LIN {X 0,Y 408.428,Z 752.813,A -85,B 0,C 180,E1 10680.84,E2 10680.84} C_VEL
LIN {X 0,Y 404.021,Z 784.174,A -85,B 0,C 180,E1 10684.706,E2 10684.706} C_VEL
LIN {X 0,Y 400.788,Z 809.614,A -85,B 0,C 180,E1 10688.967,E2 10688.967} C_VEL
LIN {X 0,Y 398.664,Z 830.61,A -85,B 0,C 180,E1 10693.733,E2 10693.733} C_VEL
LIN {X 0,Y 397.715,Z 845.382,A -85,B 0,C 180,E1 10698.469,E2 10698.469} C_VEL
LIN {X 0,Y 397.631,Z 847.747,A -85,B 0,C 180,E1 10699.458,E2 10699.458} C_VEL
LIN {X 0,Y 395.083,Z 851.309,A -85,B 0,C 180,E1 10701.251,E2 10701.251} C_VEL
LIN {X 0,Y 389.791,Z 854.941,A -85,B 0,C 180,E1 10704.007,E2 10704.007} C_VEL
LIN {X 0,Y 389.709,Z 855.317,A -85,B 0,C 180,E1 10704.327,E2 10704.327} C_VEL
LIN {X 0,Y 389.668,Z 858.175,A -85,B 0,C 180,E1 10707.771,E2 10707.771} C_VEL
LIN {X 0,Y 389.693,Z 858.182,A -85,B 0,C 180,E1 10712.225,E2 10712.225} C_VEL
LIN {X 0,Y 389.728,Z 854.056,A -85,B 0,C 180,E1 10716.691,E2 10716.691} C_VEL
LIN {X 0,Y 389.922,Z 844.142,A -85,B 0,C 180,E1 10721.76,E2 10721.76} C_VEL
LIN {X 0,Y 390.93,Z 828.247,A -85,B 0,C 180,E1 10726.884,E2 10726.884} C_VEL
LIN {X 0,Y 393.21,Z 806.828,A -85,B 0,C 180,E1 10731.751,E2 10731.751} C_VEL
LIN {X 0,Y 397.092,Z 778.974,A -85,B 0,C 180,E1 10736.349,E2 10736.349} C_VEL
LIN {X 0,Y 401.785,Z 748.417,A -85,B 0,C 180,E1 10740.034,E2 10740.034} C_VEL
LIN {X 0,Y 406.818,Z 713.375,A -85,B 0,C 180,E1 10743.071,E2 10743.071} C_VEL
LIN {X 0,Y 411.253,Z 676.937,A -85,B 0,C 180,E1 10745.194,E2 10745.194} C_VEL
LIN {X 0,Y 413.797,Z 641.889,A -85,B 0,C 180,E1 10746.487,E2 10746.487} C_VEL
LIN {X 0,Y 400.605,Z 608.761,A -85,B 0,C 180,E1 10748.579,E2 10748.579} C_VEL
LIN {X 0,Y 387.28,Z 580.66,A -85,B 0,C 180,E1 10750.746,E2 10750.746} C_VEL
LIN {X 0,Y 387.242,Z 580.66,A -85,B 0,C 180,E1 10757.972,E2 10757.972} C_VEL
LIN {X 0,Y 387.329,Z 580.66,A -85,B 0,C 180,E1 10765.168,E2 10765.168} C_VEL
LIN {X 0,Y 387.521,Z 580.66,A -85,B 0,C 180,E1 10772.048,E2 10772.048} C_VEL
LIN {X 0,Y 387.806,Z 580.66,A -85,B 0,C 180,E1 10779.543,E2 10779.543} C_VEL
LIN {X 0,Y 387.952,Z 580.66,A -85,B 0,C 180,E1 10786.464,E2 10786.464} C_VEL
LIN {X 0,Y 388.392,Z 580.66,A -85,B 0,C 180,E1 10793.29,E2 10793.29} C_VEL
LIN {X 0,Y 388.731,Z 580.66,A -85,B 0,C 180,E1 10800.006,E2 10800.006} C_VEL
LIN {X 0,Y 388.325,Z 580.66,A -85,B 0,C 180,E1 10806.723,E2 10806.723} C_VEL
LIN {X 0,Y 388.031,Z 580.66,A -85,B 0,C 180,E1 10813.546,E2 10813.546} C_VEL
LIN {X 0,Y 387.797,Z 580.66,A -85,B 0,C 180,E1 10820.578,E2 10820.578} C_VEL
LIN {X 0,Y 387.538,Z 580.66,A -85,B 0,C 180,E1 10827.964,E2 10827.964} C_VEL
LIN {X 0,Y 387.36,Z 580.66,A -85,B 0,C 180,E1 10835.902,E2 10835.902} C_VEL
LIN {X 0,Y 387.152,Z 580.66,A -85,B 0,C 180,E1 10842.013,E2 10842.013} C_VEL
LIN {X 0,Y 387.17,Z 580.66,A -85,B 0,C 180,E1 10848.337,E2 10848.337} C_VEL
LIN {X 0,Y 387.501,Z 581.204,A -85,B 0,C 180,E1 10855.685,E2 10855.685} C_VEL
LIN {X 0,Y 400.111,Z 612.182,A -85,B 0,C 180,E1 10858.859,E2 10858.859} C_VEL
LIN {X 0,Y 408.135,Z 640.7,A -85,B 0,C 180,E1 10862.182,E2 10862.182} C_VEL
LIN {X 0,Y 408.327,Z 648.198,A -85,B 0,C 180,E1 10863.018,E2 10863.018} C_VEL
LIN {X 0,Y 403.521,Z 675.315,A -85,B 0,C 180,E1 10866.233,E2 10866.233} C_VEL
LIN {X 0,Y 399.051,Z 697.721,A -85,B 0,C 180,E1 10870.036,E2 10870.036} C_VEL
LIN {X 0,Y 395.127,Z 716.014,A -85,B 0,C 180,E1 10874.444,E2 10874.444} C_VEL
LIN {X 0,Y 392.367,Z 729.811,A -85,B 0,C 180,E1 10879.554,E2 10879.554} C_VEL
LIN {X 0,Y 391.047,Z 737.35,A -85,B 0,C 180,E1 10884.448,E2 10884.448} C_VEL
LIN {X 0,Y 390.565,Z 740.223,A -85,B 0,C 180,E1 10890.002,E2 10890.002} C_VEL
LIN {X 0,Y 391.048,Z 737.251,A -85,B 0,C 180,E1 10895.557,E2 10895.557} C_VEL
LIN {X 0,Y 392.34,Z 729.704,A -85,B 0,C 180,E1 10900.402,E2 10900.402} C_VEL
LIN {X 0,Y 394.76,Z 717.487,A -85,B 0,C 180,E1 10905.006,E2 10905.006} C_VEL
LIN {X 0,Y 398.476,Z 699.978,A -85,B 0,C 180,E1 10909.42,E2 10909.42} C_VEL
LIN {X 0,Y 402.996,Z 677.934,A -85,B 0,C 180,E1 10913.277,E2 10913.277} C_VEL
LIN {X 0,Y 407.688,Z 652.329,A -85,B 0,C 180,E1 10916.467,E2 10916.467} C_VEL
LIN {X 0,Y 408.513,Z 642.184,A -85,B 0,C 180,E1 10917.525,E2 10917.525} C_VEL
LIN {X 0,Y 400.672,Z 614.076,A -85,B 0,C 180,E1 10920.832,E2 10920.832} C_VEL
LIN {X 0,Y 388.716,Z 584.955,A -85,B 0,C 180,E1 10923.905,E2 10923.905} C_VEL
LIN {X 0,Y 387.379,Z 580.66,A -85,B 0,C 180,E1 10924.312,E2 10924.312} C_VEL
LIN {X 0,Y 387.223,Z 580.66,A -85,B 0,C 180,E1 10931.661,E2 10931.661} C_VEL
LIN {X 0,Y 387.212,Z 580.66,A -85,B 0,C 180,E1 10938.331,E2 10938.331} C_VEL
LIN {X 0,Y 387.234,Z 580.66,A -85,B 0,C 180,E1 10945.195,E2 10945.195} C_VEL
LIN {X 0,Y 387.521,Z 580.66,A -85,B 0,C 180,E1 10952.034,E2 10952.034} C_VEL
LIN {X 0,Y 387.844,Z 580.66,A -85,B 0,C 180,E1 10959.54,E2 10959.54} C_VEL
LIN {X 0,Y 387.884,Z 580.66,A -85,B 0,C 180,E1 10966.449,E2 10966.449} C_VEL
LIN {X 0,Y 388.423,Z 580.66,A -85,B 0,C 180,E1 10973.278,E2 10973.278} C_VEL
LIN {X 0,Y 388.731,Z 580.66,A -85,B 0,C 180,E1 10979.994,E2 10979.994} C_VEL
LIN {X 0,Y 388.342,Z 580.66,A -85,B 0,C 180,E1 10986.71,E2 10986.71} C_VEL
LIN {X 0,Y 388.039,Z 580.66,A -85,B 0,C 180,E1 10993.532,E2 10993.532} C_VEL
LIN {X 0,Y 387.8,Z 580.66,A -85,B 0,C 180,E1 11000.565,E2 11000.565} C_VEL
LIN {X 0,Y 387.52,Z 580.66,A -85,B 0,C 180,E1 11007.952,E2 11007.952} C_VEL
LIN {X 0,Y 387.321,Z 580.66,A -85,B 0,C 180,E1 11014.824,E2 11014.824} C_VEL
LIN {X 0,Y 387.199,Z 580.66,A -85,B 0,C 180,E1 11022.015,E2 11022.015} C_VEL
LIN {X 0,Y 387.338,Z 580.66,A -85,B 0,C 180,E1 11029.326,E2 11029.326} C_VEL
LIN {X 0,Y 395.978,Z 599.127,A -85,B 0,C 180,E1 11030.728,E2 11030.728} C_VEL
LIN {X 0,Y 411.678,Z 635.468,A -85,B 0,C 180,E1 11033.137,E2 11033.137} C_VEL
LIN {X 0,Y 414.185,Z 645.901,A -85,B 0,C 180,E1 11033.687,E2 11033.687} C_VEL
LIN {X 0,Y 410.314,Z 684.949,A -85,B 0,C 180,E1 11035.193,E2 11035.193} C_VEL
LIN {X 0,Y 405.769,Z 720.46,A -85,B 0,C 180,E1 11037.462,E2 11037.462} C_VEL
LIN {X 0,Y 400.817,Z 754.356,A -85,B 0,C 180,E1 11040.588,E2 11040.588} C_VEL
LIN {X 0,Y 396.311,Z 784.649,A -85,B 0,C 180,E1 11044.482,E2 11044.482} C_VEL
LIN {X 0,Y 392.955,Z 809.701,A -85,B 0,C 180,E1 11048.823,E2 11048.823} C_VEL
LIN {X 0,Y 390.795,Z 830.377,A -85,B 0,C 180,E1 11053.685,E2 11053.685} C_VEL
LIN {X 0,Y 389.827,Z 845.492,A -85,B 0,C 180,E1 11058.8,E2 11058.8} C_VEL
LIN {X 0,Y 389.735,Z 854.049,A -85,B 0,C 180,E1 11063.305,E2 11063.305} C_VEL
LIN {X 0,Y 389.709,Z 855.317,A -85,B 0,C 180,E1 11064.327,E2 11064.327} C_VEL
LIN {X 0,Y 387.19,Z 856.88,A -85,B 0,C 180,E1 11066.212,E2 11066.212} C_VEL
LIN {X 0,Y 381.917,Z 857.427,A -85,B 0,C 180,E1 11069.077,E2 11069.077} C_VEL
LIN {X 0,Y 381.856,Z 857.421,A -85,B 0,C 180,E1 11069.408,E2 11069.408} C_VEL
LIN {X 0,Y 381.884,Z 855.425,A -85,B 0,C 180,E1 11074.546,E2 11074.546} C_VEL
LIN {X 0,Y 381.91,Z 849.075,A -85,B 0,C 180,E1 11079.122,E2 11079.122} C_VEL
LIN {X 0,Y 382.441,Z 836.232,A -85,B 0,C 180,E1 11084.44,E2 11084.44} C_VEL
LIN {X 0,Y 384.2,Z 817.301,A -85,B 0,C 180,E1 11089.683,E2 11089.683} C_VEL
LIN {X 0,Y 387.498,Z 792.723,A -85,B 0,C 180,E1 11094.526,E2 11094.526} C_VEL
LIN {X 0,Y 391.958,Z 763.881,A -85,B 0,C 180,E1 11098.711,E2 11098.711} C_VEL
LIN {X 0,Y 397.257,Z 730.096,A -85,B 0,C 180,E1 11102.244,E2 11102.244} C_VEL
LIN {X 0,Y 402.324,Z 695.108,A -85,B 0,C 180,E1 11104.795,E2 11104.795} C_VEL
LIN {X 0,Y 406.63,Z 657.105,A -85,B 0,C 180,E1 11106.562,E2 11106.562} C_VEL
LIN {X 0,Y 407.134,Z 644.103,A -85,B 0,C 180,E1 11107.017,E2 11107.017} C_VEL
LIN {X 0,Y 394.189,Z 611.589,A -85,B 0,C 180,E1 11109.175,E2 11109.175} C_VEL
LIN {X 0,Y 379.324,Z 580.66,A -85,B 0,C 180,E1 11111.638,E2 11111.638} C_VEL
LIN {X 0,Y 379.285,Z 580.66,A -85,B 0,C 180,E1 11117.274,E2 11117.274} C_VEL
LIN {X 0,Y 379.32,Z 580.66,A -85,B 0,C 180,E1 11123.23,E2 11123.23} C_VEL
LIN {X 0,Y 379.421,Z 580.66,A -85,B 0,C 180,E1 11128.759,E2 11128.759} C_VEL
LIN {X 0,Y 379.685,Z 580.66,A -85,B 0,C 180,E1 11136.506,E2 11136.506} C_VEL
LIN {X 0,Y 379.941,Z 580.66,A -85,B 0,C 180,E1 11143.809,E2 11143.809} C_VEL
LIN {X 0,Y 380.271,Z 580.66,A -85,B 0,C 180,E1 11150.843,E2 11150.843} C_VEL
LIN {X 0,Y 380.781,Z 580.66,A -85,B 0,C 180,E1 11157.728,E2 11157.728} C_VEL
LIN {X 0,Y 380.595,Z 580.66,A -85,B 0,C 180,E1 11164.57,E2 11164.57} C_VEL
LIN {X 0,Y 380.168,Z 580.66,A -85,B 0,C 180,E1 11171.492,E2 11171.492} C_VEL
LIN {X 0,Y 379.949,Z 580.66,A -85,B 0,C 180,E1 11178.596,E2 11178.596} C_VEL
LIN {X 0,Y 379.641,Z 580.66,A -85,B 0,C 180,E1 11186.027,E2 11186.027} C_VEL
LIN {X 0,Y 379.449,Z 580.66,A -85,B 0,C 180,E1 11193.967,E2 11193.967} C_VEL
LIN {X 0,Y 379.2,Z 580.66,A -85,B 0,C 180,E1 11200.662,E2 11200.662} C_VEL
LIN {X 0,Y 379.165,Z 580.66,A -85,B 0,C 180,E1 11207.252,E2 11207.252} C_VEL
LIN {X 0,Y 379.517,Z 580.66,A -85,B 0,C 180,E1 11214.699,E2 11214.699} C_VEL
LIN {X 0,Y 392.526,Z 612.432,A -85,B 0,C 180,E1 11218.068,E2 11218.068} C_VEL
LIN {X 0,Y 400.461,Z 640.281,A -85,B 0,C 180,E1 11221.385,E2 11221.385} C_VEL
LIN {X 0,Y 401.55,Z 648.886,A -85,B 0,C 180,E1 11222.445,E2 11222.445} C_VEL
LIN {X 0,Y 396.58,Z 675.766,A -85,B 0,C 180,E1 11225.66,E2 11225.66} C_VEL
LIN {X 0,Y 391.704,Z 698.972,A -85,B 0,C 180,E1 11229.645,E2 11229.645} C_VEL
LIN {X 0,Y 387.601,Z 717.228,A -85,B 0,C 180,E1 11234.134,E2 11234.134} C_VEL
LIN {X 0,Y 384.971,Z 729.548,A -85,B 0,C 180,E1 11238.662,E2 11238.662} C_VEL
LIN {X 0,Y 383.57,Z 737.237,A -85,B 0,C 180,E1 11243.201,E2 11243.201} C_VEL
LIN {X 0,Y 382.888,Z 740.919,A -85,B 0,C 180,E1 11247.736,E2 11247.736} C_VEL
LIN {X 0,Y 383,Z 740.86,A -85,B 0,C 180,E1 11252.268,E2 11252.268} C_VEL
LIN {X 0,Y 383.558,Z 737.112,A -85,B 0,C 180,E1 11256.803,E2 11256.803} C_VEL
LIN {X 0,Y 385.296,Z 728.075,A -85,B 0,C 180,E1 11261.908,E2 11261.908} C_VEL
LIN {X 0,Y 388.46,Z 713.123,A -85,B 0,C 180,E1 11266.937,E2 11266.937} C_VEL
LIN {X 0,Y 392.989,Z 692.75,A -85,B 0,C 180,E1 11271.471,E2 11271.471} C_VEL
LIN {X 0,Y 397.941,Z 668.776,A -85,B 0,C 180,E1 11275.194,E2 11275.194} C_VEL
LIN {X 0,Y 401.712,Z 645.578,A -85,B 0,C 180,E1 11277.822,E2 11277.822} C_VEL
LIN {X 0,Y 394.415,Z 618.304,A -85,B 0,C 180,E1 11281.162,E2 11281.162} C_VEL
LIN {X 0,Y 383.249,Z 590.025,A -85,B 0,C 180,E1 11284.285,E2 11284.285} C_VEL
LIN {X 0,Y 379.427,Z 580.66,A -85,B 0,C 180,E1 11285.311,E2 11285.311} C_VEL
LIN {X 0,Y 379.232,Z 580.66,A -85,B 0,C 180,E1 11292.745,E2 11292.745} C_VEL
LIN {X 0,Y 379.221,Z 580.66,A -85,B 0,C 180,E1 11300.29,E2 11300.29} C_VEL
LIN {X 0,Y 379.372,Z 580.66,A -85,B 0,C 180,E1 11306.942,E2 11306.942} C_VEL
LIN {X 0,Y 379.642,Z 580.66,A -85,B 0,C 180,E1 11313.973,E2 11313.973} C_VEL
LIN {X 0,Y 379.927,Z 580.66,A -85,B 0,C 180,E1 11321.403,E2 11321.403} C_VEL
LIN {X 0,Y 380.06,Z 580.66,A -85,B 0,C 180,E1 11328.504,E2 11328.504} C_VEL
LIN {X 0,Y 380.542,Z 580.66,A -85,B 0,C 180,E1 11335.43,E2 11335.43} C_VEL
LIN {X 0,Y 380.829,Z 580.66,A -85,B 0,C 180,E1 11339.994,E2 11339.994} C_VEL
LIN {X 0,Y 380.431,Z 580.66,A -85,B 0,C 180,E1 11346.851,E2 11346.851} C_VEL
LIN {X 0,Y 380.096,Z 580.66,A -85,B 0,C 180,E1 11353.821,E2 11353.821} C_VEL
LIN {X 0,Y 379.823,Z 580.66,A -85,B 0,C 180,E1 11361.017,E2 11361.017} C_VEL
LIN {X 0,Y 379.537,Z 580.66,A -85,B 0,C 180,E1 11368.641,E2 11368.641} C_VEL
LIN {X 0,Y 379.402,Z 580.66,A -85,B 0,C 180,E1 11373.957,E2 11373.957} C_VEL
LIN {X 0,Y 379.234,Z 580.66,A -85,B 0,C 180,E1 11380.661,E2 11380.661} C_VEL
LIN {X 0,Y 379.354,Z 580.66,A -85,B 0,C 180,E1 11388.357,E2 11388.357} C_VEL
LIN {X 0,Y 402.366,Z 630.289,A -85,B 0,C 180,E1 11392.12,E2 11392.12} C_VEL
LIN {X 0,Y 407.505,Z 646.855,A -85,B 0,C 180,E1 11393.118,E2 11393.118} C_VEL
LIN {X 0,Y 403.389,Z 685.45,A -85,B 0,C 180,E1 11394.662,E2 11394.662} C_VEL
LIN {X 0,Y 398.627,Z 720.792,A -85,B 0,C 180,E1 11396.983,E2 11396.983} C_VEL
LIN {X 0,Y 393.277,Z 755.365,A -85,B 0,C 180,E1 11400.285,E2 11400.285} C_VEL
LIN {X 0,Y 388.564,Z 785.437,A -85,B 0,C 180,E1 11404.295,E2 11404.295} C_VEL
LIN {X 0,Y 384.994,Z 811.22,A -85,B 0,C 180,E1 11408.97,E2 11408.97} C_VEL
LIN {X 0,Y 382.809,Z 831.032,A -85,B 0,C 180,E1 11413.925,E2 11413.925} C_VEL
LIN {X 0,Y 381.942,Z 845.542,A -85,B 0,C 180,E1 11419.145,E2 11419.145} C_VEL
LIN {X 0,Y 381.903,Z 854.237,A -85,B 0,C 180,E1 11424.31,E2 11424.31} C_VEL
LIN {X 0,Y 381.856,Z 857.421,A -85,B 0,C 180,E1 11429.408,E2 11429.408} C_VEL
LIN {X 0,Y 379.393,Z 857.009,A -85,B 0,C 180,E1 11431.343,E2 11431.343} C_VEL
LIN {X 0,Y 374.108,Z 854.57,A -85,B 0,C 180,E1 11434.246,E2 11434.246} C_VEL
LIN {X 0,Y 374.055,Z 854.268,A -85,B 0,C 180,E1 11434.584,E2 11434.584} C_VEL
LIN {X 0,Y 374.058,Z 847.85,A -85,B 0,C 180,E1 11439.315,E2 11439.315} C_VEL
LIN {X 0,Y 374.602,Z 835.485,A -85,B 0,C 180,E1 11444.569,E2 11444.569} C_VEL
LIN {X 0,Y 376.472,Z 816.475,A -85,B 0,C 180,E1 11449.987,E2 11449.987} C_VEL
LIN {X 0,Y 380.035,Z 791.361,A -85,B 0,C 180,E1 11455.04,E2 11455.04} C_VEL
LIN {X 0,Y 384.927,Z 761.75,A -85,B 0,C 180,E1 11459.388,E2 11459.388} C_VEL
LIN {X 0,Y 390.339,Z 728.546,A -85,B 0,C 180,E1 11462.887,E2 11462.887} C_VEL
LIN {X 0,Y 395.823,Z 692.6,A -85,B 0,C 180,E1 11465.513,E2 11465.513} C_VEL
LIN {X 0,Y 400.25,Z 654.842,A -85,B 0,C 180,E1 11467.243,E2 11467.243} C_VEL
LIN {X 0,Y 400.059,Z 644.9,A -85,B 0,C 180,E1 11467.658,E2 11467.658} C_VEL
LIN {X 0,Y 386.799,Z 612.231,A -85,B 0,C 180,E1 11469.957,E2 11469.957} C_VEL
LIN {X 0,Y 371.426,Z 581.632,A -85,B 0,C 180,E1 11472.55,E2 11472.55} C_VEL
LIN {X 0,Y 371.358,Z 580.66,A -85,B 0,C 180,E1 11472.799,E2 11472.799} C_VEL
LIN {X 0,Y 371.392,Z 580.66,A -85,B 0,C 180,E1 11479.296,E2 11479.296} C_VEL
LIN {X 0,Y 371.383,Z 580.66,A -85,B 0,C 180,E1 11485.206,E2 11485.206} C_VEL
LIN {X 0,Y 371.544,Z 580.66,A -85,B 0,C 180,E1 11490.733,E2 11490.733} C_VEL
LIN {X 0,Y 371.713,Z 580.66,A -85,B 0,C 180,E1 11495.971,E2 11495.971} C_VEL
LIN {X 0,Y 371.943,Z 580.66,A -85,B 0,C 180,E1 11501.002,E2 11501.002} C_VEL
LIN {X 0,Y 372.142,Z 580.66,A -85,B 0,C 180,E1 11508.27,E2 11508.27} C_VEL
LIN {X 0,Y 372.599,Z 580.66,A -85,B 0,C 180,E1 11515.345,E2 11515.345} C_VEL
LIN {X 0,Y 372.928,Z 580.66,A -85,B 0,C 180,E1 11520.006,E2 11520.006} C_VEL
LIN {X 0,Y 372.487,Z 580.66,A -85,B 0,C 180,E1 11527.011,E2 11527.011} C_VEL
LIN {X 0,Y 372.146,Z 580.66,A -85,B 0,C 180,E1 11534.135,E2 11534.135} C_VEL
LIN {X 0,Y 371.841,Z 580.66,A -85,B 0,C 180,E1 11541.504,E2 11541.504} C_VEL
LIN {X 0,Y 371.647,Z 580.66,A -85,B 0,C 180,E1 11546.63,E2 11546.63} C_VEL
LIN {X 0,Y 371.531,Z 580.66,A -85,B 0,C 180,E1 11551.997,E2 11551.997} C_VEL
LIN {X 0,Y 371.314,Z 580.66,A -85,B 0,C 180,E1 11559.224,E2 11559.224} C_VEL
LIN {X 0,Y 371.241,Z 580.66,A -85,B 0,C 180,E1 11566.111,E2 11566.111} C_VEL
LIN {X 0,Y 371.502,Z 580.66,A -85,B 0,C 180,E1 11573.68,E2 11573.68} C_VEL
LIN {X 0,Y 385.033,Z 612.913,A -85,B 0,C 180,E1 11577.267,E2 11577.267} C_VEL
LIN {X 0,Y 393.296,Z 641.778,A -85,B 0,C 180,E1 11580.814,E2 11580.814} C_VEL
LIN {X 0,Y 394.422,Z 651.706,A -85,B 0,C 180,E1 11582.07,E2 11582.07} C_VEL
LIN {X 0,Y 389.345,Z 677.782,A -85,B 0,C 180,E1 11585.292,E2 11585.292} C_VEL
LIN {X 0,Y 384.395,Z 700.217,A -85,B 0,C 180,E1 11589.24,E2 11589.24} C_VEL
LIN {X 0,Y 380.07,Z 718.443,A -85,B 0,C 180,E1 11593.811,E2 11593.811} C_VEL
LIN {X 0,Y 376.989,Z 732.207,A -85,B 0,C 180,E1 11599.12,E2 11599.12} C_VEL
LIN {X 0,Y 375.503,Z 739.727,A -85,B 0,C 180,E1 11604.217,E2 11604.217} C_VEL
LIN {X 0,Y 374.961,Z 742.594,A -85,B 0,C 180,E1 11610.002,E2 11610.002} C_VEL
LIN {X 0,Y 375.362,Z 740.704,A -85,B 0,C 180,E1 11614.629,E2 11614.629} C_VEL
LIN {X 0,Y 376.741,Z 733.236,A -85,B 0,C 180,E1 11620.241,E2 11620.241} C_VEL
LIN {X 0,Y 379.285,Z 721.716,A -85,B 0,C 180,E1 11625.04,E2 11625.04} C_VEL
LIN {X 0,Y 383.507,Z 703.74,A -85,B 0,C 180,E1 11629.91,E2 11629.91} C_VEL
LIN {X 0,Y 388.481,Z 681.784,A -85,B 0,C 180,E1 11633.988,E2 11633.988} C_VEL
LIN {X 0,Y 393.842,Z 655.099,A -85,B 0,C 180,E1 11637.474,E2 11637.474} C_VEL
LIN {X 0,Y 394.48,Z 647.059,A -85,B 0,C 180,E1 11638.38,E2 11638.38} C_VEL
LIN {X 0,Y 387.275,Z 619.827,A -85,B 0,C 180,E1 11641.82,E2 11641.82} C_VEL
LIN {X 0,Y 376.077,Z 591.221,A -85,B 0,C 180,E1 11645.09,E2 11645.09} C_VEL
LIN {X 0,Y 371.464,Z 580.66,A -85,B 0,C 180,E1 11646.202,E2 11646.202} C_VEL
LIN {X 0,Y 371.317,Z 580.66,A -85,B 0,C 180,E1 11653.884,E2 11653.884} C_VEL
LIN {X 0,Y 371.291,Z 580.66,A -85,B 0,C 180,E1 11660.787,E2 11660.787} C_VEL
LIN {X 0,Y 371.46,Z 580.66,A -85,B 0,C 180,E1 11667.996,E2 11667.996} C_VEL
LIN {X 0,Y 371.689,Z 580.66,A -85,B 0,C 180,E1 11673.66,E2 11673.66} C_VEL
LIN {X 0,Y 371.964,Z 580.66,A -85,B 0,C 180,E1 11680.989,E2 11680.989} C_VEL
LIN {X 0,Y 372.117,Z 580.66,A -85,B 0,C 180,E1 11688.255,E2 11688.255} C_VEL
LIN {X 0,Y 372.63,Z 580.66,A -85,B 0,C 180,E1 11695.332,E2 11695.332} C_VEL
LIN {X 0,Y 372.927,Z 580.66,A -85,B 0,C 180,E1 11699.994,E2 11699.994} C_VEL
LIN {X 0,Y 372.504,Z 580.66,A -85,B 0,C 180,E1 11706.997,E2 11706.997} C_VEL
LIN {X 0,Y 372.153,Z 580.66,A -85,B 0,C 180,E1 11714.122,E2 11714.122} C_VEL
LIN {X 0,Y 371.848,Z 580.66,A -85,B 0,C 180,E1 11721.49,E2 11721.49} C_VEL
LIN {X 0,Y 371.664,Z 580.66,A -85,B 0,C 180,E1 11726.615,E2 11726.615} C_VEL
LIN {X 0,Y 371.492,Z 580.66,A -85,B 0,C 180,E1 11731.986,E2 11731.986} C_VEL
LIN {X 0,Y 371.293,Z 580.66,A -85,B 0,C 180,E1 11739.213,E2 11739.213} C_VEL
LIN {X 0,Y 371.346,Z 580.66,A -85,B 0,C 180,E1 11746.12,E2 11746.12} C_VEL
LIN {X 0,Y 371.418,Z 581.101,A -85,B 0,C 180,E1 11747.451,E2 11747.451} C_VEL
LIN {X 0,Y 394.617,Z 629.646,A -85,B 0,C 180,E1 11751.327,E2 11751.327} C_VEL
LIN {X 0,Y 400.779,Z 648.749,A -85,B 0,C 180,E1 11752.559,E2 11752.559} C_VEL
LIN {X 0,Y 396.475,Z 686.244,A -85,B 0,C 180,E1 11754.129,E2 11754.129} C_VEL
LIN {X 0,Y 391.426,Z 721.858,A -85,B 0,C 180,E1 11756.546,E2 11756.546} C_VEL
LIN {X 0,Y 385.878,Z 755.621,A -85,B 0,C 180,E1 11759.883,E2 11759.883} C_VEL
LIN {X 0,Y 381.114,Z 784.292,A -85,B 0,C 180,E1 11763.796,E2 11763.796} C_VEL
LIN {X 0,Y 377.281,Z 810.188,A -85,B 0,C 180,E1 11768.588,E2 11768.588} C_VEL
LIN {X 0,Y 375.061,Z 829.759,A -85,B 0,C 180,E1 11773.584,E2 11773.584} C_VEL
LIN {X 0,Y 374.088,Z 844.302,A -85,B 0,C 180,E1 11778.914,E2 11778.914} C_VEL
LIN {X 0,Y 374.059,Z 851.627,A -85,B 0,C 180,E1 11783.023,E2 11783.023} C_VEL
LIN {X 0,Y 374.022,Z 855.793,A -85,B 0,C 180,E1 11787.678,E2 11787.678} C_VEL
LIN {X 0,Y 374.046,Z 855.8,A -85,B 0,C 180,E1 11792.318,E2 11792.318} C_VEL
LIN {X 0,Y 374.055,Z 854.268,A -85,B 0,C 180,E1 11794.584,E2 11794.584} C_VEL
LIN {X 0,Y 371.675,Z 852.023,A -85,B 0,C 180,E1 11796.532,E2 11796.532} C_VEL
LIN {X 0,Y 366.191,Z 846.21,A -85,B 0,C 180,E1 11799.745,E2 11799.745} C_VEL
LIN {X 0,Y 366.784,Z 834.049,A -85,B 0,C 180,E1 11804.949,E2 11804.949} C_VEL
LIN {X 0,Y 368.788,Z 815.171,A -85,B 0,C 180,E1 11810.421,E2 11810.421} C_VEL
LIN {X 0,Y 372.296,Z 791.726,A -85,B 0,C 180,E1 11815.275,E2 11815.275} C_VEL
LIN {X 0,Y 377.3,Z 762.964,A -85,B 0,C 180,E1 11819.654,E2 11819.654} C_VEL
LIN {X 0,Y 382.986,Z 730.216,A -85,B 0,C 180,E1 11823.262,E2 11823.262} C_VEL
LIN {X 0,Y 388.518,Z 695.78,A -85,B 0,C 180,E1 11825.9,E2 11825.9} C_VEL
LIN {X 0,Y 393.056,Z 660.377,A -85,B 0,C 180,E1 11827.677,E2 11827.677} C_VEL
LIN {X 0,Y 393.679,Z 647.851,A -85,B 0,C 180,E1 11828.175,E2 11828.175} C_VEL
LIN {X 0,Y 380.811,Z 615.816,A -85,B 0,C 180,E1 11830.543,E2 11830.543} C_VEL
LIN {X 0,Y 363.49,Z 581.418,A -85,B 0,C 180,E1 11833.589,E2 11833.589} C_VEL
LIN {X 0,Y 363.437,Z 580.66,A -85,B 0,C 180,E1 11838.574,E2 11838.574} C_VEL
LIN {X 0,Y 363.416,Z 580.66,A -85,B 0,C 180,E1 11844.329,E2 11844.329} C_VEL
LIN {X 0,Y 363.633,Z 580.66,A -85,B 0,C 180,E1 11850.964,E2 11850.964} C_VEL
LIN {X 0,Y 363.852,Z 580.66,A -85,B 0,C 180,E1 11858.014,E2 11858.014} C_VEL
LIN {X 0,Y 364.13,Z 580.66,A -85,B 0,C 180,E1 11865.56,E2 11865.56} C_VEL
LIN {X 0,Y 364.637,Z 580.66,A -85,B 0,C 180,E1 11872.851,E2 11872.851} C_VEL
LIN {X 0,Y 365.026,Z 580.66,A -85,B 0,C 180,E1 11880.007,E2 11880.007} C_VEL
LIN {X 0,Y 364.565,Z 580.66,A -85,B 0,C 180,E1 11887.164,E2 11887.164} C_VEL
LIN {X 0,Y 364.203,Z 580.66,A -85,B 0,C 180,E1 11894.45,E2 11894.45} C_VEL
LIN {X 0,Y 363.857,Z 580.66,A -85,B 0,C 180,E1 11902,E2 11902} C_VEL
LIN {X 0,Y 363.648,Z 580.66,A -85,B 0,C 180,E1 11909.982,E2 11909.982} C_VEL
LIN {X 0,Y 363.432,Z 580.66,A -85,B 0,C 180,E1 11917.676,E2 11917.676} C_VEL
LIN {X 0,Y 363.298,Z 580.66,A -85,B 0,C 180,E1 11925.12,E2 11925.12} C_VEL
LIN {X 0,Y 363.485,Z 580.66,A -85,B 0,C 180,E1 11932.622,E2 11932.622} C_VEL
LIN {X 0,Y 377.063,Z 611.983,A -85,B 0,C 180,E1 11936.263,E2 11936.263} C_VEL
LIN {X 0,Y 385.452,Z 640.208,A -85,B 0,C 180,E1 11939.797,E2 11939.797} C_VEL
LIN {X 0,Y 387.493,Z 653.618,A -85,B 0,C 180,E1 11941.589,E2 11941.589} C_VEL
LIN {X 0,Y 381.967,Z 680.428,A -85,B 0,C 180,E1 11945.017,E2 11945.017} C_VEL
LIN {X 0,Y 376.775,Z 702.827,A -85,B 0,C 180,E1 11949.109,E2 11949.109} C_VEL
LIN {X 0,Y 372.137,Z 721.447,A -85,B 0,C 180,E1 11954.063,E2 11954.063} C_VEL
LIN {X 0,Y 369.095,Z 734.296,A -85,B 0,C 180,E1 11959.366,E2 11959.366} C_VEL
LIN {X 0,Y 367.581,Z 741.975,A -85,B 0,C 180,E1 11965.277,E2 11965.277} C_VEL
LIN {X 0,Y 367.151,Z 743.78,A -85,B 0,C 180,E1 11970.002,E2 11970.002} C_VEL
LIN {X 0,Y 367.585,Z 741.892,A -85,B 0,C 180,E1 11974.727,E2 11974.727} C_VEL
LIN {X 0,Y 369.089,Z 734.318,A -85,B 0,C 180,E1 11980.52,E2 11980.52} C_VEL
LIN {X 0,Y 372.174,Z 721.133,A -85,B 0,C 180,E1 11985.94,E2 11985.94} C_VEL
LIN {X 0,Y 376.474,Z 703.725,A -85,B 0,C 180,E1 11990.605,E2 11990.605} C_VEL
LIN {X 0,Y 381.596,Z 682.072,A -85,B 0,C 180,E1 11994.621,E2 11994.621} C_VEL
LIN {X 0,Y 386.962,Z 656.461,A -85,B 0,C 180,E1 11998.005,E2 11998.005} C_VEL
LIN {X 0,Y 387.378,Z 649.091,A -85,B 0,C 180,E1 11998.877,E2 11998.877} C_VEL
LIN {X 0,Y 380.233,Z 621.505,A -85,B 0,C 180,E1 12002.483,E2 12002.483} C_VEL
LIN {X 0,Y 369.012,Z 593.381,A -85,B 0,C 180,E1 12005.867,E2 12005.867} C_VEL
LIN {X 0,Y 363.447,Z 580.66,A -85,B 0,C 180,E1 12007.273,E2 12007.273} C_VEL
LIN {X 0,Y 363.409,Z 580.66,A -85,B 0,C 180,E1 12011.807,E2 12011.807} C_VEL
LIN {X 0,Y 363.408,Z 580.66,A -85,B 0,C 180,E1 12018.586,E2 12018.586} C_VEL
LIN {X 0,Y 363.348,Z 580.66,A -85,B 0,C 180,E1 12024.304,E2 12024.304} C_VEL
LIN {X 0,Y 363.654,Z 580.66,A -85,B 0,C 180,E1 12030.967,E2 12030.967} C_VEL
LIN {X 0,Y 363.883,Z 580.66,A -85,B 0,C 180,E1 12038.001,E2 12038.001} C_VEL
LIN {X 0,Y 364.094,Z 580.66,A -85,B 0,C 180,E1 12045.545,E2 12045.545} C_VEL
LIN {X 0,Y 364.667,Z 580.66,A -85,B 0,C 180,E1 12052.838,E2 12052.838} C_VEL
LIN {X 0,Y 365.025,Z 580.66,A -85,B 0,C 180,E1 12059.993,E2 12059.993} C_VEL
LIN {X 0,Y 364.582,Z 580.66,A -85,B 0,C 180,E1 12067.15,E2 12067.15} C_VEL
LIN {X 0,Y 364.209,Z 580.66,A -85,B 0,C 180,E1 12074.436,E2 12074.436} C_VEL
LIN {X 0,Y 363.868,Z 580.66,A -85,B 0,C 180,E1 12081.985,E2 12081.985} C_VEL
LIN {X 0,Y 363.624,Z 580.66,A -85,B 0,C 180,E1 12089.969,E2 12089.969} C_VEL
LIN {X 0,Y 363.388,Z 580.66,A -85,B 0,C 180,E1 12097.66,E2 12097.66} C_VEL
LIN {X 0,Y 363.38,Z 580.66,A -85,B 0,C 180,E1 12105.088,E2 12105.088} C_VEL
LIN {X 0,Y 363.455,Z 581.03,A -85,B 0,C 180,E1 12106.414,E2 12106.414} C_VEL
LIN {X 0,Y 386.913,Z 629.264,A -85,B 0,C 180,E1 12110.506,E2 12110.506} C_VEL
LIN {X 0,Y 394.032,Z 650.612,A -85,B 0,C 180,E1 12111.99,E2 12111.99} C_VEL
LIN {X 0,Y 389.63,Z 686.73,A -85,B 0,C 180,E1 12113.558,E2 12113.558} C_VEL
LIN {X 0,Y 384.113,Z 723.58,A -85,B 0,C 180,E1 12116.154,E2 12116.154} C_VEL
LIN {X 0,Y 378.31,Z 756.824,A -85,B 0,C 180,E1 12119.579,E2 12119.579} C_VEL
LIN {X 0,Y 373.132,Z 786.486,A -85,B 0,C 180,E1 12123.813,E2 12123.813} C_VEL
LIN {X 0,Y 369.324,Z 811.204,A -85,B 0,C 180,E1 12128.662,E2 12128.662} C_VEL
LIN {X 0,Y 367.073,Z 830.408,A -85,B 0,C 180,E1 12133.833,E2 12133.833} C_VEL
LIN {X 0,Y 366.199,Z 844.357,A -85,B 0,C 180,E1 12139.275,E2 12139.275} C_VEL
LIN {X 0,Y 366.241,Z 851.831,A -85,B 0,C 180,E1 12144.066,E2 12144.066} C_VEL
LIN {X 0,Y 366.198,Z 854.602,A -85,B 0,C 180,E1 12147.628,E2 12147.628} C_VEL
LIN {X 0,Y 366.221,Z 854.61,A -85,B 0,C 180,E1 12152.367,E2 12152.367} C_VEL
LIN {X 0,Y 366.22,Z 850.3,A -85,B 0,C 180,E1 12157.21,E2 12157.21} C_VEL
LIN {X 0,Y 366.191,Z 846.21,A -85,B 0,C 180,E1 12159.745,E2 12159.745} C_VEL
LIN {X 0,Y 364.976,Z 843.6,A -85,B 0,C 180,E1 12161.041,E2 12161.041} C_VEL
LIN {X 0,Y 358.924,Z 834.938,A -85,B 0,C 180,E1 12164.507,E2 12164.507} C_VEL
LIN {X 0,Y 358.888,Z 834.042,A -85,B 0,C 180,E1 12164.829,E2 12164.829} C_VEL
LIN {X 0,Y 360.804,Z 816.272,A -85,B 0,C 180,E1 12170.252,E2 12170.252} C_VEL
LIN {X 0,Y 364.574,Z 792.097,A -85,B 0,C 180,E1 12175.52,E2 12175.52} C_VEL
LIN {X 0,Y 369.631,Z 764.368,A -85,B 0,C 180,E1 12179.906,E2 12179.906} C_VEL
LIN {X 0,Y 375.623,Z 731.825,A -85,B 0,C 180,E1 12183.654,E2 12183.654} C_VEL
LIN {X 0,Y 381.531,Z 697.189,A -85,B 0,C 180,E1 12186.413,E2 12186.413} C_VEL
LIN {X 0,Y 386.341,Z 661.576,A -85,B 0,C 180,E1 12188.273,E2 12188.273} C_VEL
LIN {X 0,Y 386.913,Z 649.803,A -85,B 0,C 180,E1 12188.772,E2 12188.772} C_VEL
LIN {X 0,Y 374.847,Z 619.227,A -85,B 0,C 180,E1 12191.155,E2 12191.155} C_VEL
LIN {X 0,Y 355.507,Z 581.275,A -85,B 0,C 180,E1 12194.697,E2 12194.697} C_VEL
LIN {X 0,Y 355.428,Z 580.66,A -85,B 0,C 180,E1 12200.295,E2 12200.295} C_VEL
LIN {X 0,Y 355.522,Z 580.66,A -85,B 0,C 180,E1 12206.393,E2 12206.393} C_VEL
LIN {X 0,Y 355.733,Z 580.66,A -85,B 0,C 180,E1 12213.346,E2 12213.346} C_VEL
LIN {X 0,Y 356.042,Z 580.66,A -85,B 0,C 180,E1 12220.119,E2 12220.119} C_VEL
LIN {X 0,Y 356.305,Z 580.66,A -85,B 0,C 180,E1 12227.764,E2 12227.764} C_VEL
LIN {X 0,Y 356.798,Z 580.66,A -85,B 0,C 180,E1 12235.138,E2 12235.138} C_VEL
LIN {X 0,Y 357.137,Z 580.66,A -85,B 0,C 180,E1 12240.007,E2 12240.007} C_VEL
LIN {X 0,Y 356.634,Z 580.66,A -85,B 0,C 180,E1 12247.324,E2 12247.324} C_VEL
LIN {X 0,Y 356.259,Z 580.66,A -85,B 0,C 180,E1 12254.78,E2 12254.78} C_VEL
LIN {X 0,Y 355.904,Z 580.66,A -85,B 0,C 180,E1 12262.518,E2 12262.518} C_VEL
LIN {X 0,Y 355.754,Z 580.66,A -85,B 0,C 180,E1 12267.921,E2 12267.921} C_VEL
LIN {X 0,Y 355.525,Z 580.66,A -85,B 0,C 180,E1 12275.993,E2 12275.993} C_VEL
LIN {X 0,Y 355.298,Z 580.66,A -85,B 0,C 180,E1 12283.583,E2 12283.583} C_VEL
LIN {X 0,Y 355.547,Z 581.262,A -85,B 0,C 180,E1 12291.538,E2 12291.538} C_VEL
LIN {X 0,Y 369.328,Z 611.913,A -85,B 0,C 180,E1 12295.298,E2 12295.298} C_VEL
LIN {X 0,Y 377.475,Z 638.181,A -85,B 0,C 180,E1 12298.692,E2 12298.692} C_VEL
LIN {X 0,Y 380.604,Z 655.399,A -85,B 0,C 180,E1 12301.076,E2 12301.076} C_VEL
LIN {X 0,Y 374.823,Z 682.16,A -85,B 0,C 180,E1 12304.587,E2 12304.587} C_VEL
LIN {X 0,Y 369.493,Z 704.068,A -85,B 0,C 180,E1 12308.677,E2 12308.677} C_VEL
LIN {X 0,Y 364.605,Z 722.661,A -85,B 0,C 180,E1 12313.725,E2 12313.725} C_VEL
LIN {X 0,Y 361.423,Z 735.487,A -85,B 0,C 180,E1 12319.137,E2 12319.137} C_VEL
LIN {X 0,Y 359.789,Z 743.164,A -85,B 0,C 180,E1 12325.174,E2 12325.174} C_VEL
LIN {X 0,Y 359.358,Z 744.964,A -85,B 0,C 180,E1 12330.002,E2 12330.002} C_VEL
LIN {X 0,Y 359.793,Z 743.082,A -85,B 0,C 180,E1 12334.83,E2 12334.83} C_VEL
LIN {X 0,Y 361.457,Z 735.307,A -85,B 0,C 180,E1 12340.867,E2 12340.867} C_VEL
LIN {X 0,Y 364.645,Z 722.35,A -85,B 0,C 180,E1 12346.278,E2 12346.278} C_VEL
LIN {X 0,Y 369.185,Z 704.964,A -85,B 0,C 180,E1 12351.031,E2 12351.031} C_VEL
LIN {X 0,Y 374.54,Z 683.349,A -85,B 0,C 180,E1 12355.118,E2 12355.118} C_VEL
LIN {X 0,Y 380.321,Z 656.837,A -85,B 0,C 180,E1 12358.666,E2 12358.666} C_VEL
LIN {X 0,Y 380.064,Z 649.804,A -85,B 0,C 180,E1 12359.586,E2 12359.586} C_VEL
LIN {X 0,Y 373.011,Z 622.548,A -85,B 0,C 180,E1 12363.255,E2 12363.255} C_VEL
LIN {X 0,Y 361.91,Z 594.917,A -85,B 0,C 180,E1 12366.725,E2 12366.725} C_VEL
LIN {X 0,Y 355.532,Z 580.66,A -85,B 0,C 180,E1 12368.465,E2 12368.465} C_VEL
LIN {X 0,Y 355.348,Z 580.66,A -85,B 0,C 180,E1 12376.415,E2 12376.415} C_VEL
LIN {X 0,Y 355.45,Z 580.66,A -85,B 0,C 180,E1 12384.031,E2 12384.031} C_VEL
LIN {X 0,Y 355.724,Z 580.66,A -85,B 0,C 180,E1 12392.076,E2 12392.076} C_VEL
LIN {X 0,Y 356.064,Z 580.66,A -85,B 0,C 180,E1 12400.106,E2 12400.106} C_VEL
LIN {X 0,Y 356.289,Z 580.66,A -85,B 0,C 180,E1 12407.797,E2 12407.797} C_VEL
LIN {X 0,Y 356.833,Z 580.66,A -85,B 0,C 180,E1 12415.125,E2 12415.125} C_VEL
LIN {X 0,Y 357.136,Z 580.66,A -85,B 0,C 180,E1 12419.993,E2 12419.993} C_VEL
LIN {X 0,Y 356.651,Z 580.66,A -85,B 0,C 180,E1 12427.31,E2 12427.31} C_VEL
LIN {X 0,Y 356.264,Z 580.66,A -85,B 0,C 180,E1 12434.766,E2 12434.766} C_VEL
LIN {X 0,Y 355.924,Z 580.66,A -85,B 0,C 180,E1 12442.502,E2 12442.502} C_VEL
LIN {X 0,Y 355.748,Z 580.66,A -85,B 0,C 180,E1 12447.906,E2 12447.906} C_VEL
LIN {X 0,Y 355.477,Z 580.66,A -85,B 0,C 180,E1 12455.975,E2 12455.975} C_VEL
LIN {X 0,Y 355.36,Z 580.66,A -85,B 0,C 180,E1 12463.587,E2 12463.587} C_VEL
LIN {X 0,Y 355.487,Z 580.66,A -85,B 0,C 180,E1 12465.3,E2 12465.3} C_VEL
LIN {X 0,Y 359.96,Z 590.459,A -85,B 0,C 180,E1 12466.201,E2 12466.201} C_VEL
LIN {X 0,Y 378.966,Z 628.21,A -85,B 0,C 180,E1 12469.594,E2 12469.594} C_VEL
LIN {X 0,Y 387.3,Z 652.392,A -85,B 0,C 180,E1 12471.394,E2 12471.394} C_VEL
LIN {X 0,Y 382.535,Z 689.924,A -85,B 0,C 180,E1 12473.127,E2 12473.127} C_VEL
LIN {X 0,Y 376.744,Z 725.352,A -85,B 0,C 180,E1 12475.76,E2 12475.76} C_VEL
LIN {X 0,Y 370.724,Z 758.203,A -85,B 0,C 180,E1 12479.282,E2 12479.282} C_VEL
LIN {X 0,Y 365.436,Z 786.857,A -85,B 0,C 180,E1 12483.55,E2 12483.55} C_VEL
LIN {X 0,Y 361.498,Z 811.207,A -85,B 0,C 180,E1 12488.5,E2 12488.5} C_VEL
LIN {X 0,Y 359.111,Z 831.047,A -85,B 0,C 180,E1 12494.093,E2 12494.093} C_VEL
LIN {X 0,Y 358.335,Z 844.292,A -85,B 0,C 180,E1 12499.653,E2 12499.653} C_VEL
LIN {X 0,Y 358.43,Z 850.823,A -85,B 0,C 180,E1 12504.105,E2 12504.105} C_VEL
LIN {X 0,Y 358.507,Z 854.015,A -85,B 0,C 180,E1 12509.998,E2 12509.998} C_VEL
LIN {X 0,Y 358.405,Z 851.837,A -85,B 0,C 180,E1 12514.844,E2 12514.844} C_VEL
LIN {X 0,Y 358.346,Z 845.403,A -85,B 0,C 180,E1 12519.727,E2 12519.727} C_VEL
LIN {X 0,Y 358.888,Z 834.042,A -85,B 0,C 180,E1 12524.829,E2 12524.829} C_VEL
LIN {X 0,Y 355.532,Z 826.744,A -85,B 0,C 180,E1 12527.332,E2 12527.332} C_VEL
LIN {X 0,Y 352.605,Z 818.428,A -85,B 0,C 180,E1 12529.795,E2 12529.795} C_VEL
LIN {X 0,Y 356.198,Z 795.555,A -85,B 0,C 180,E1 12535.151,E2 12535.151} C_VEL
LIN {X 0,Y 361.699,Z 767.163,A -85,B 0,C 180,E1 12539.977,E2 12539.977} C_VEL
LIN {X 0,Y 367.984,Z 734.707,A -85,B 0,C 180,E1 12543.916,E2 12543.916} C_VEL
LIN {X 0,Y 374.341,Z 699.923,A -85,B 0,C 180,E1 12546.859,E2 12546.859} C_VEL
LIN {X 0,Y 379.575,Z 663.79,A -85,B 0,C 180,E1 12548.846,E2 12548.846} C_VEL
LIN {X 0,Y 380.304,Z 652.031,A -85,B 0,C 180,E1 12549.367,E2 12549.367} C_VEL
LIN {X 0,Y 368.171,Z 621.085,A -85,B 0,C 180,E1 12551.921,E2 12551.921} C_VEL
LIN {X 0,Y 349.383,Z 585.742,A -85,B 0,C 180,E1 12555.462,E2 12555.462} C_VEL
LIN {X 0,Y 347.491,Z 580.66,A -85,B 0,C 180,E1 12556.078,E2 12556.078} C_VEL
LIN {X 0,Y 347.446,Z 580.66,A -85,B 0,C 180,E1 12562.415,E2 12562.415} C_VEL
LIN {X 0,Y 347.641,Z 580.66,A -85,B 0,C 180,E1 12568.5,E2 12568.5} C_VEL
LIN {X 0,Y 347.837,Z 580.66,A -85,B 0,C 180,E1 12576.067,E2 12576.067} C_VEL
LIN {X 0,Y 348.255,Z 580.66,A -85,B 0,C 180,E1 12583.018,E2 12583.018} C_VEL
LIN {X 0,Y 348.506,Z 580.66,A -85,B 0,C 180,E1 12590,E2 12590} C_VEL
LIN {X 0,Y 349.142,Z 580.66,A -85,B 0,C 180,E1 12597.522,E2 12597.522} C_VEL
LIN {X 0,Y 348.984,Z 580.66,A -85,B 0,C 180,E1 12603.816,E2 12603.816} C_VEL
LIN {X 0,Y 348.557,Z 580.66,A -85,B 0,C 180,E1 12610.013,E2 12610.013} C_VEL
LIN {X 0,Y 348.261,Z 580.66,A -85,B 0,C 180,E1 12617.724,E2 12617.724} C_VEL
LIN {X 0,Y 347.835,Z 580.66,A -85,B 0,C 180,E1 12625.81,E2 12625.81} C_VEL
LIN {X 0,Y 347.678,Z 580.66,A -85,B 0,C 180,E1 12631.512,E2 12631.512} C_VEL
LIN {X 0,Y 347.421,Z 580.66,A -85,B 0,C 180,E1 12638.337,E2 12638.337} C_VEL
LIN {X 0,Y 347.327,Z 580.66,A -85,B 0,C 180,E1 12645.78,E2 12645.78} C_VEL
LIN {X 0,Y 347.545,Z 581.129,A -85,B 0,C 180,E1 12650.337,E2 12650.337} C_VEL
LIN {X 0,Y 361.954,Z 612.44,A -85,B 0,C 180,E1 12654.374,E2 12654.374} C_VEL
LIN {X 0,Y 370.13,Z 638.684,A -85,B 0,C 180,E1 12657.878,E2 12657.878} C_VEL
LIN {X 0,Y 373.483,Z 658.435,A -85,B 0,C 180,E1 12660.683,E2 12660.683} C_VEL
LIN {X 0,Y 367.337,Z 685.261,A -85,B 0,C 180,E1 12664.359,E2 12664.359} C_VEL
LIN {X 0,Y 361.537,Z 707.858,A -85,B 0,C 180,E1 12668.829,E2 12668.829} C_VEL
LIN {X 0,Y 356.652,Z 725.656,A -85,B 0,C 180,E1 12673.985,E2 12673.985} C_VEL
LIN {X 0,Y 353.496,Z 737.719,A -85,B 0,C 180,E1 12679.514,E2 12679.514} C_VEL
LIN {X 0,Y 352.015,Z 744.349,A -85,B 0,C 180,E1 12685.068,E2 12685.068} C_VEL
LIN {X 0,Y 351.549,Z 746.15,A -85,B 0,C 180,E1 12690.002,E2 12690.002} C_VEL
LIN {X 0,Y 352.019,Z 744.27,A -85,B 0,C 180,E1 12694.937,E2 12694.937} C_VEL
LIN {X 0,Y 353.783,Z 736.502,A -85,B 0,C 180,E1 12701.106,E2 12701.106} C_VEL
LIN {X 0,Y 357.145,Z 723.562,A -85,B 0,C 180,E1 12706.63,E2 12706.63} C_VEL
LIN {X 0,Y 361.907,Z 706.201,A -85,B 0,C 180,E1 12711.475,E2 12711.475} C_VEL
LIN {X 0,Y 367.508,Z 684.631,A -85,B 0,C 180,E1 12715.633,E2 12715.633} C_VEL
LIN {X 0,Y 373.334,Z 659.156,A -85,B 0,C 180,E1 12719.123,E2 12719.123} C_VEL
LIN {X 0,Y 372.303,Z 648.184,A -85,B 0,C 180,E1 12720.661,E2 12720.661} C_VEL
LIN {X 0,Y 365.082,Z 621.24,A -85,B 0,C 180,E1 12724.364,E2 12724.364} C_VEL
LIN {X 0,Y 353.277,Z 593.168,A -85,B 0,C 180,E1 12728.053,E2 12728.053} C_VEL
LIN {X 0,Y 347.606,Z 581.673,A -85,B 0,C 180,E1 12729.512,E2 12729.512} C_VEL
LIN {X 0,Y 347.551,Z 580.66,A -85,B 0,C 180,E1 12729.664,E2 12729.664} C_VEL
LIN {X 0,Y 347.374,Z 580.66,A -85,B 0,C 180,E1 12737.815,E2 12737.815} C_VEL
LIN {X 0,Y 347.53,Z 580.66,A -85,B 0,C 180,E1 12745.871,E2 12745.871} C_VEL
LIN {X 0,Y 347.706,Z 580.66,A -85,B 0,C 180,E1 12751.374,E2 12751.374} C_VEL
LIN {X 0,Y 347.934,Z 580.66,A -85,B 0,C 180,E1 12756.936,E2 12756.936} C_VEL
LIN {X 0,Y 348.213,Z 580.66,A -85,B 0,C 180,E1 12763.057,E2 12763.057} C_VEL
LIN {X 0,Y 348.508,Z 580.66,A -85,B 0,C 180,E1 12769.986,E2 12769.986} C_VEL
LIN {X 0,Y 349.173,Z 580.66,A -85,B 0,C 180,E1 12777.508,E2 12777.508} C_VEL
LIN {X 0,Y 348.948,Z 580.66,A -85,B 0,C 180,E1 12784.971,E2 12784.971} C_VEL
LIN {X 0,Y 348.48,Z 580.66,A -85,B 0,C 180,E1 12792.539,E2 12792.539} C_VEL
LIN {X 0,Y 348.266,Z 580.66,A -85,B 0,C 180,E1 12797.71,E2 12797.71} C_VEL
LIN {X 0,Y 347.842,Z 580.66,A -85,B 0,C 180,E1 12805.794,E2 12805.794} C_VEL
LIN {X 0,Y 347.644,Z 580.66,A -85,B 0,C 180,E1 12811.499,E2 12811.499} C_VEL
LIN {X 0,Y 347.398,Z 580.66,A -85,B 0,C 180,E1 12818.325,E2 12818.325} C_VEL
LIN {X 0,Y 347.488,Z 580.66,A -85,B 0,C 180,E1 12824.121,E2 12824.121} C_VEL
LIN {X 0,Y 350.155,Z 586.523,A -85,B 0,C 180,E1 12824.698,E2 12824.698} C_VEL
LIN {X 0,Y 370.68,Z 626.494,A -85,B 0,C 180,E1 12828.569,E2 12828.569} C_VEL
LIN {X 0,Y 380.681,Z 653.364,A -85,B 0,C 180,E1 12830.747,E2 12830.747} C_VEL
LIN {X 0,Y 375.645,Z 691.055,A -85,B 0,C 180,E1 12832.568,E2 12832.568} C_VEL
LIN {X 0,Y 369.733,Z 725.427,A -85,B 0,C 180,E1 12835.196,E2 12835.196} C_VEL
LIN {X 0,Y 363.494,Z 757.913,A -85,B 0,C 180,E1 12838.766,E2 12838.766} C_VEL
LIN {X 0,Y 357.691,Z 787.491,A -85,B 0,C 180,E1 12843.323,E2 12843.323} C_VEL
LIN {X 0,Y 353.498,Z 812.528,A -85,B 0,C 180,E1 12848.648,E2 12848.648} C_VEL
LIN {X 0,Y 351.155,Z 831.509,A -85,B 0,C 180,E1 12854.365,E2 12854.365} C_VEL
LIN {X 0,Y 350.493,Z 844.168,A -85,B 0,C 180,E1 12860.048,E2 12860.048} C_VEL
LIN {X 0,Y 350.576,Z 850.633,A -85,B 0,C 180,E1 12865.043,E2 12865.043} C_VEL
LIN {X 0,Y 350.693,Z 852.828,A -85,B 0,C 180,E1 12869.998,E2 12869.998} C_VEL
LIN {X 0,Y 350.582,Z 850.643,A -85,B 0,C 180,E1 12874.953,E2 12874.953} C_VEL
LIN {X 0,Y 350.503,Z 844.183,A -85,B 0,C 180,E1 12879.947,E2 12879.947} C_VEL
LIN {X 0,Y 351.182,Z 831.537,A -85,B 0,C 180,E1 12885.629,E2 12885.629} C_VEL
LIN {X 0,Y 352.605,Z 818.428,A -85,B 0,C 180,E1 12889.795,E2 12889.795} C_VEL
LIN {X 0,Y 350.001,Z 809.418,A -85,B 0,C 180,E1 12892.205,E2 12892.205} C_VEL
LIN {X 0,Y 347.693,Z 799.669,A -85,B 0,C 180,E1 12894.586,E2 12894.586} C_VEL
LIN {X 0,Y 353.23,Z 771.93,A -85,B 0,C 180,E1 12899.706,E2 12899.706} C_VEL
LIN {X 0,Y 359.547,Z 741.687,A -85,B 0,C 180,E1 12903.73,E2 12903.73} C_VEL
LIN {X 0,Y 366.067,Z 708.718,A -85,B 0,C 180,E1 12906.846,E2 12906.846} C_VEL
LIN {X 0,Y 371.751,Z 673.442,A -85,B 0,C 180,E1 12909.087,E2 12909.087} C_VEL
LIN {X 0,Y 373.72,Z 654.128,A -85,B 0,C 180,E1 12909.991,E2 12909.991} C_VEL
LIN {X 0,Y 361.373,Z 622.626,A -85,B 0,C 180,E1 12912.738,E2 12912.738} C_VEL
LIN {X 0,Y 341.857,Z 586.188,A -85,B 0,C 180,E1 12916.607,E2 12916.607} C_VEL
LIN {X 0,Y 339.541,Z 580.66,A -85,B 0,C 180,E1 12917.314,E2 12917.314} C_VEL
LIN {X 0,Y 339.519,Z 580.66,A -85,B 0,C 180,E1 12924.578,E2 12924.578} C_VEL
LIN {X 0,Y 339.782,Z 580.66,A -85,B 0,C 180,E1 12930.658,E2 12930.658} C_VEL
LIN {X 0,Y 340.123,Z 580.66,A -85,B 0,C 180,E1 12939.188,E2 12939.188} C_VEL
LIN {X 0,Y 340.401,Z 580.66,A -85,B 0,C 180,E1 12947.158,E2 12947.158} C_VEL
LIN {X 0,Y 340.976,Z 580.66,A -85,B 0,C 180,E1 12954.912,E2 12954.912} C_VEL
LIN {X 0,Y 341.347,Z 580.66,A -85,B 0,C 180,E1 12960.007,E2 12960.007} C_VEL
LIN {X 0,Y 340.777,Z 580.66,A -85,B 0,C 180,E1 12967.667,E2 12967.667} C_VEL
LIN {X 0,Y 340.377,Z 580.66,A -85,B 0,C 180,E1 12975.486,E2 12975.486} C_VEL
LIN {X 0,Y 340.142,Z 580.66,A -85,B 0,C 180,E1 12980.868,E2 12980.868} C_VEL
LIN {X 0,Y 339.809,Z 580.66,A -85,B 0,C 180,E1 12989.356,E2 12989.356} C_VEL
LIN {X 0,Y 339.489,Z 580.66,A -85,B 0,C 180,E1 12996.611,E2 12996.611} C_VEL
LIN {X 0,Y 339.44,Z 580.66,A -85,B 0,C 180,E1 13004.47,E2 13004.47} C_VEL
LIN {X 0,Y 339.496,Z 580.945,A -85,B 0,C 180,E1 13009.046,E2 13009.046} C_VEL
LIN {X 0,Y 344.265,Z 590.944,A -85,B 0,C 180,E1 13010.331,E2 13010.331} C_VEL
LIN {X 0,Y 356.56,Z 618.174,A -85,B 0,C 180,E1 13014.102,E2 13014.102} C_VEL
LIN {X 0,Y 364.32,Z 645.294,A -85,B 0,C 180,E1 13017.917,E2 13017.917} C_VEL
LIN {X 0,Y 366.526,Z 660.543,A -85,B 0,C 180,E1 13020.178,E2 13020.178} C_VEL
LIN {X 0,Y 360.321,Z 686.536,A -85,B 0,C 180,E1 13023.822,E2 13023.822} C_VEL
LIN {X 0,Y 354.275,Z 709.082,A -85,B 0,C 180,E1 13028.373,E2 13028.373} C_VEL
LIN {X 0,Y 349.128,Z 726.863,A -85,B 0,C 180,E1 13033.63,E2 13033.63} C_VEL
LIN {X 0,Y 345.816,Z 738.912,A -85,B 0,C 180,E1 13039.279,E2 13039.279} C_VEL
LIN {X 0,Y 344.227,Z 745.537,A -85,B 0,C 180,E1 13044.956,E2 13044.956} C_VEL
LIN {X 0,Y 343.763,Z 747.333,A -85,B 0,C 180,E1 13050.002,E2 13050.002} C_VEL
LIN {X 0,Y 344.231,Z 745.459,A -85,B 0,C 180,E1 13055.049,E2 13055.049} C_VEL
LIN {X 0,Y 346.102,Z 737.699,A -85,B 0,C 180,E1 13061.355,E2 13061.355} C_VEL
LIN {X 0,Y 349.644,Z 724.776,A -85,B 0,C 180,E1 13066.997,E2 13066.997} C_VEL
LIN {X 0,Y 355.028,Z 706.091,A -85,B 0,C 180,E1 13072.242,E2 13072.242} C_VEL
LIN {X 0,Y 360.93,Z 684.094,A -85,B 0,C 180,E1 13076.47,E2 13076.47} C_VEL
LIN {X 0,Y 366.823,Z 658.992,A -85,B 0,C 180,E1 13079.903,E2 13079.903} C_VEL
LIN {X 0,Y 361.193,Z 632.932,A -85,B 0,C 180,E1 13083.748,E2 13083.748} C_VEL
LIN {X 0,Y 351.631,Z 606.094,A -85,B 0,C 180,E1 13087.438,E2 13087.438} C_VEL
LIN {X 0,Y 339.573,Z 581.581,A -85,B 0,C 180,E1 13090.792,E2 13090.792} C_VEL
LIN {X 0,Y 339.478,Z 580.66,A -85,B 0,C 180,E1 13091.298,E2 13091.298} C_VEL
LIN {X 0,Y 339.465,Z 580.66,A -85,B 0,C 180,E1 13098,E2 13098} C_VEL
LIN {X 0,Y 339.459,Z 580.66,A -85,B 0,C 180,E1 13104.554,E2 13104.554} C_VEL
LIN {X 0,Y 339.756,Z 580.66,A -85,B 0,C 180,E1 13110.639,E2 13110.639} C_VEL
LIN {X 0,Y 340.162,Z 580.66,A -85,B 0,C 180,E1 13119.184,E2 13119.184} C_VEL
LIN {X 0,Y 340.398,Z 580.66,A -85,B 0,C 180,E1 13127.143,E2 13127.143} C_VEL
LIN {X 0,Y 341.011,Z 580.66,A -85,B 0,C 180,E1 13134.899,E2 13134.899} C_VEL
LIN {X 0,Y 341.346,Z 580.66,A -85,B 0,C 180,E1 13139.993,E2 13139.993} C_VEL
LIN {X 0,Y 340.793,Z 580.66,A -85,B 0,C 180,E1 13147.652,E2 13147.652} C_VEL
LIN {X 0,Y 340.388,Z 580.66,A -85,B 0,C 180,E1 13155.471,E2 13155.471} C_VEL
LIN {X 0,Y 340.141,Z 580.66,A -85,B 0,C 180,E1 13160.853,E2 13160.853} C_VEL
LIN {X 0,Y 339.792,Z 580.66,A -85,B 0,C 180,E1 13169.341,E2 13169.341} C_VEL
LIN {X 0,Y 339.454,Z 580.66,A -85,B 0,C 180,E1 13176.595,E2 13176.595} C_VEL
LIN {X 0,Y 339.562,Z 580.66,A -85,B 0,C 180,E1 13182.854,E2 13182.854} C_VEL
LIN {X 0,Y 342.133,Z 586.47,A -85,B 0,C 180,E1 13183.471,E2 13183.471} C_VEL
LIN {X 0,Y 362.229,Z 624.421,A -85,B 0,C 180,E1 13187.448,E2 13187.448} C_VEL
LIN {X 0,Y 373.997,Z 655.285,A -85,B 0,C 180,E1 13190.109,E2 13190.109} C_VEL
LIN {X 0,Y 368.785,Z 692.165,A -85,B 0,C 180,E1 13191.986,E2 13191.986} C_VEL
LIN {X 0,Y 362.454,Z 727.106,A -85,B 0,C 180,E1 13194.76,E2 13194.76} C_VEL
LIN {X 0,Y 355.795,Z 759.652,A -85,B 0,C 180,E1 13198.509,E2 13198.509} C_VEL
LIN {X 0,Y 349.926,Z 788.29,A -85,B 0,C 180,E1 13203.116,E2 13203.116} C_VEL
LIN {X 0,Y 345.69,Z 812.453,A -85,B 0,C 180,E1 13208.479,E2 13208.479} C_VEL
LIN {X 0,Y 343.371,Z 830.253,A -85,B 0,C 180,E1 13214.001,E2 13214.001} C_VEL
LIN {X 0,Y 342.64,Z 842.945,A -85,B 0,C 180,E1 13219.817,E2 13219.817} C_VEL
LIN {X 0,Y 342.768,Z 849.44,A -85,B 0,C 180,E1 13224.929,E2 13224.929} C_VEL
LIN {X 0,Y 342.878,Z 851.641,A -85,B 0,C 180,E1 13229.998,E2 13229.998} C_VEL
LIN {X 0,Y 342.772,Z 849.45,A -85,B 0,C 180,E1 13235.066,E2 13235.066} C_VEL
LIN {X 0,Y 342.651,Z 842.961,A -85,B 0,C 180,E1 13240.178,E2 13240.178} C_VEL
LIN {X 0,Y 343.385,Z 830.282,A -85,B 0,C 180,E1 13245.993,E2 13245.993} C_VEL
LIN {X 0,Y 345.816,Z 811.265,A -85,B 0,C 180,E1 13251.845,E2 13251.845} C_VEL
LIN {X 0,Y 347.693,Z 799.669,A -85,B 0,C 180,E1 13254.586,E2 13254.586} C_VEL
LIN {X 0,Y 345.917,Z 789.294,A -85,B 0,C 180,E1 13256.907,E2 13256.907} C_VEL
LIN {X 0,Y 344.498,Z 778.067,A -85,B 0,C 180,E1 13259.135,E2 13259.135} C_VEL
LIN {X 0,Y 351.074,Z 748.637,A -85,B 0,C 180,E1 13263.463,E2 13263.463} C_VEL
LIN {X 0,Y 357.813,Z 715.998,A -85,B 0,C 180,E1 13266.89,E2 13266.89} C_VEL
LIN {X 0,Y 364.212,Z 679.782,A -85,B 0,C 180,E1 13269.46,E2 13269.46} C_VEL
LIN {X 0,Y 367.023,Z 655.882,A -85,B 0,C 180,E1 13270.66,E2 13270.66} C_VEL
LIN {X 0,Y 354.12,Z 623.133,A -85,B 0,C 180,E1 13273.694,E2 13273.694} C_VEL
LIN {X 0,Y 335.897,Z 589.69,A -85,B 0,C 180,E1 13277.469,E2 13277.469} C_VEL
LIN {X 0,Y 331.634,Z 581.396,A -85,B 0,C 180,E1 13278.458,E2 13278.458} C_VEL
LIN {X 0,Y 331.574,Z 580.66,A -85,B 0,C 180,E1 13285.272,E2 13285.272} C_VEL
LIN {X 0,Y 331.89,Z 580.66,A -85,B 0,C 180,E1 13292.867,E2 13292.867} C_VEL
LIN {X 0,Y 332.26,Z 580.66,A -85,B 0,C 180,E1 13301.407,E2 13301.407} C_VEL
LIN {X 0,Y 332.622,Z 580.66,A -85,B 0,C 180,E1 13309.517,E2 13309.517} C_VEL
LIN {X 0,Y 333.325,Z 580.66,A -85,B 0,C 180,E1 13317.404,E2 13317.404} C_VEL
LIN {X 0,Y 333.328,Z 580.66,A -85,B 0,C 180,E1 13322.611,E2 13322.611} C_VEL
LIN {X 0,Y 332.691,Z 580.66,A -85,B 0,C 180,E1 13330.496,E2 13330.496} C_VEL
LIN {X 0,Y 332.307,Z 580.66,A -85,B 0,C 180,E1 13338.606,E2 13338.606} C_VEL
LIN {X 0,Y 331.905,Z 580.66,A -85,B 0,C 180,E1 13347.148,E2 13347.148} C_VEL
LIN {X 0,Y 331.606,Z 580.66,A -85,B 0,C 180,E1 13354.736,E2 13354.736} C_VEL
LIN {X 0,Y 331.535,Z 580.66,A -85,B 0,C 180,E1 13359.752,E2 13359.752} C_VEL
LIN {X 0,Y 331.516,Z 580.784,A -85,B 0,C 180,E1 13367.675,E2 13367.675} C_VEL
LIN {X 0,Y 334.05,Z 586.434,A -85,B 0,C 180,E1 13368.397,E2 13368.397} C_VEL
LIN {X 0,Y 347.184,Z 613.654,A -85,B 0,C 180,E1 13372.376,E2 13372.376} C_VEL
LIN {X 0,Y 355.564,Z 639.231,A -85,B 0,C 180,E1 13376.081,E2 13376.081} C_VEL
LIN {X 0,Y 359.857,Z 660.735,A -85,B 0,C 180,E1 13379.396,E2 13379.396} C_VEL
LIN {X 0,Y 353.345,Z 687.808,A -85,B 0,C 180,E1 13383.265,E2 13383.265} C_VEL
LIN {X 0,Y 347.021,Z 710.308,A -85,B 0,C 180,E1 13387.898,E2 13387.898} C_VEL
LIN {X 0,Y 341.627,Z 728.067,A -85,B 0,C 180,E1 13393.26,E2 13393.26} C_VEL
LIN {X 0,Y 338.128,Z 740.107,A -85,B 0,C 180,E1 13399.032,E2 13399.032} C_VEL
LIN {X 0,Y 336.457,Z 746.722,A -85,B 0,C 180,E1 13404.839,E2 13404.839} C_VEL
LIN {X 0,Y 335.954,Z 748.519,A -85,B 0,C 180,E1 13410.002,E2 13410.002} C_VEL
LIN {X 0,Y 336.461,Z 746.646,A -85,B 0,C 180,E1 13415.166,E2 13415.166} C_VEL
LIN {X 0,Y 338.453,Z 738.891,A -85,B 0,C 180,E1 13421.615,E2 13421.615} C_VEL
LIN {X 0,Y 342.166,Z 725.987,A -85,B 0,C 180,E1 13427.38,E2 13427.38} C_VEL
LIN {X 0,Y 347.81,Z 707.332,A -85,B 0,C 180,E1 13432.729,E2 13432.729} C_VEL
LIN {X 0,Y 353.987,Z 685.369,A -85,B 0,C 180,E1 13437.031,E2 13437.031} C_VEL
LIN {X 0,Y 359.808,Z 660.407,A -85,B 0,C 180,E1 13440.548,E2 13440.548} C_VEL
LIN {X 0,Y 354.251,Z 634.565,A -85,B 0,C 180,E1 13444.501,E2 13444.501} C_VEL
LIN {X 0,Y 344.562,Z 607.523,A -85,B 0,C 180,E1 13448.392,E2 13448.392} C_VEL
LIN {X 0,Y 331.682,Z 582.033,A -85,B 0,C 180,E1 13452.114,E2 13452.114} C_VEL
LIN {X 0,Y 331.534,Z 580.66,A -85,B 0,C 180,E1 13452.408,E2 13452.408} C_VEL
LIN {X 0,Y 331.533,Z 580.66,A -85,B 0,C 180,E1 13460.248,E2 13460.248} C_VEL
LIN {X 0,Y 331.579,Z 580.66,A -85,B 0,C 180,E1 13466.766,E2 13466.766} C_VEL
LIN {X 0,Y 331.89,Z 580.66,A -85,B 0,C 180,E1 13472.851,E2 13472.851} C_VEL
LIN {X 0,Y 332.144,Z 580.66,A -85,B 0,C 180,E1 13478.605,E2 13478.605} C_VEL
LIN {X 0,Y 332.342,Z 580.66,A -85,B 0,C 180,E1 13484.129,E2 13484.129} C_VEL
LIN {X 0,Y 332.905,Z 580.66,A -85,B 0,C 180,E1 13492.151,E2 13492.151} C_VEL
LIN {X 0,Y 333.442,Z 580.66,A -85,B 0,C 180,E1 13499.993,E2 13499.993} C_VEL
LIN {X 0,Y 332.872,Z 580.66,A -85,B 0,C 180,E1 13507.835,E2 13507.835} C_VEL
LIN {X 0,Y 332.428,Z 580.66,A -85,B 0,C 180,E1 13515.851,E2 13515.851} C_VEL
LIN {X 0,Y 332.147,Z 580.66,A -85,B 0,C 180,E1 13521.379,E2 13521.379} C_VEL
LIN {X 0,Y 331.813,Z 580.66,A -85,B 0,C 180,E1 13529.89,E2 13529.89} C_VEL
LIN {X 0,Y 331.574,Z 580.66,A -85,B 0,C 180,E1 13536.404,E2 13536.404} C_VEL
LIN {X 0,Y 331.559,Z 580.763,A -85,B 0,C 180,E1 13541.538,E2 13541.538} C_VEL
LIN {X 0,Y 334.078,Z 586.424,A -85,B 0,C 180,E1 13542.152,E2 13542.152} C_VEL
LIN {X 0,Y 352.91,Z 620.612,A -85,B 0,C 180,E1 13546.077,E2 13546.077} C_VEL
LIN {X 0,Y 366.321,Z 653.666,A -85,B 0,C 180,E1 13549.154,E2 13549.154} C_VEL
LIN {X 0,Y 367.193,Z 659.763,A -85,B 0,C 180,E1 13549.595,E2 13549.595} C_VEL
LIN {X 0,Y 361.503,Z 695.949,A -85,B 0,C 180,E1 13551.559,E2 13551.559} C_VEL
LIN {X 0,Y 354.741,Z 730.97,A -85,B 0,C 180,E1 13554.542,E2 13554.542} C_VEL
LIN {X 0,Y 348.076,Z 761.634,A -85,B 0,C 180,E1 13558.284,E2 13558.284} C_VEL
LIN {X 0,Y 341.853,Z 790.679,A -85,B 0,C 180,E1 13563.223,E2 13563.223} C_VEL
LIN {X 0,Y 337.63,Z 813.544,A -85,B 0,C 180,E1 13568.63,E2 13568.63} C_VEL
LIN {X 0,Y 335.399,Z 830.712,A -85,B 0,C 180,E1 13574.283,E2 13574.283} C_VEL
LIN {X 0,Y 334.779,Z 842.818,A -85,B 0,C 180,E1 13580.234,E2 13580.234} C_VEL
LIN {X 0,Y 334.937,Z 848.243,A -85,B 0,C 180,E1 13584.811,E2 13584.811} C_VEL
LIN {X 0,Y 335.063,Z 850.454,A -85,B 0,C 180,E1 13589.998,E2 13589.998} C_VEL
LIN {X 0,Y 334.883,Z 847.541,A -85,B 0,C 180,E1 13596.007,E2 13596.007} C_VEL
LIN {X 0,Y 334.843,Z 839.453,A -85,B 0,C 180,E1 13601.738,E2 13601.738} C_VEL
LIN {X 0,Y 335.892,Z 825.353,A -85,B 0,C 180,E1 13607.711,E2 13607.711} C_VEL
LIN {X 0,Y 338.868,Z 806.015,A -85,B 0,C 180,E1 13613.358,E2 13613.358} C_VEL
LIN {X 0,Y 343.982,Z 780.649,A -85,B 0,C 180,E1 13618.688,E2 13618.688} C_VEL
LIN {X 0,Y 344.498,Z 778.067,A -85,B 0,C 180,E1 13619.135,E2 13619.135} C_VEL
LIN {X 0,Y 343.478,Z 766.334,A -85,B 0,C 180,E1 13621.305,E2 13621.305} C_VEL
LIN {X 0,Y 342.742,Z 753.838,A -85,B 0,C 180,E1 13623.352,E2 13623.352} C_VEL
LIN {X 0,Y 349.853,Z 721.361,A -85,B 0,C 180,E1 13627.059,E2 13627.059} C_VEL
LIN {X 0,Y 356.912,Z 684.793,A -85,B 0,C 180,E1 13629.887,E2 13629.887} C_VEL
LIN {X 0,Y 360.496,Z 658.236,A -85,B 0,C 180,E1 13631.293,E2 13631.293} C_VEL
LIN {X 0,Y 348.038,Z 626.146,A -85,B 0,C 180,E1 13634.451,E2 13634.451} C_VEL
LIN {X 0,Y 329.79,Z 592.314,A -85,B 0,C 180,E1 13638.43,E2 13638.43} C_VEL
LIN {X 0,Y 323.739,Z 581.734,A -85,B 0,C 180,E1 13639.877,E2 13639.877} C_VEL
LIN {X 0,Y 323.684,Z 580.66,A -85,B 0,C 180,E1 13640.211,E2 13640.211} C_VEL
LIN {X 0,Y 323.665,Z 580.66,A -85,B 0,C 180,E1 13647.346,E2 13647.346} C_VEL
LIN {X 0,Y 323.987,Z 580.66,A -85,B 0,C 180,E1 13655.137,E2 13655.137} C_VEL
LIN {X 0,Y 324.28,Z 580.66,A -85,B 0,C 180,E1 13660.932,E2 13660.932} C_VEL
LIN {X 0,Y 324.671,Z 580.66,A -85,B 0,C 180,E1 13669.257,E2 13669.257} C_VEL
LIN {X 0,Y 325.405,Z 580.66,A -85,B 0,C 180,E1 13677.341,E2 13677.341} C_VEL
LIN {X 0,Y 325.41,Z 580.66,A -85,B 0,C 180,E1 13682.674,E2 13682.674} C_VEL
LIN {X 0,Y 324.744,Z 580.66,A -85,B 0,C 180,E1 13690.756,E2 13690.756} C_VEL
LIN {X 0,Y 324.321,Z 580.66,A -85,B 0,C 180,E1 13699.081,E2 13699.081} C_VEL
LIN {X 0,Y 323.997,Z 580.66,A -85,B 0,C 180,E1 13707.4,E2 13707.4} C_VEL
LIN {X 0,Y 323.694,Z 580.66,A -85,B 0,C 180,E1 13714.153,E2 13714.153} C_VEL
LIN {X 0,Y 323.467,Z 580.66,A -85,B 0,C 180,E1 13721.509,E2 13721.509} C_VEL
LIN {X 0,Y 323.523,Z 580.877,A -85,B 0,C 180,E1 13726.208,E2 13726.208} C_VEL
LIN {X 0,Y 325.982,Z 586.318,A -85,B 0,C 180,E1 13726.938,E2 13726.938} C_VEL
LIN {X 0,Y 339.768,Z 613.984,A -85,B 0,C 180,E1 13731.257,E2 13731.257} C_VEL
LIN {X 0,Y 348.369,Z 639.729,A -85,B 0,C 180,E1 13735.148,E2 13735.148} C_VEL
LIN {X 0,Y 352.892,Z 663.997,A -85,B 0,C 180,E1 13739.016,E2 13739.016} C_VEL
LIN {X 0,Y 345.934,Z 690.876,A -85,B 0,C 180,E1 13742.997,E2 13742.997} C_VEL
LIN {X 0,Y 339.407,Z 712.775,A -85,B 0,C 180,E1 13747.721,E2 13747.721} C_VEL
LIN {X 0,Y 334.13,Z 729.271,A -85,B 0,C 180,E1 13752.873,E2 13752.873} C_VEL
LIN {X 0,Y 330.439,Z 741.303,A -85,B 0,C 180,E1 13758.774,E2 13758.774} C_VEL
LIN {X 0,Y 328.672,Z 747.909,A -85,B 0,C 180,E1 13764.716,E2 13764.716} C_VEL
LIN {X 0,Y 328.144,Z 749.706,A -85,B 0,C 180,E1 13770.002,E2 13770.002} C_VEL
LIN {X 0,Y 328.676,Z 747.835,A -85,B 0,C 180,E1 13775.288,E2 13775.288} C_VEL
LIN {X 0,Y 330.8,Z 740.084,A -85,B 0,C 180,E1 13781.888,E2 13781.888} C_VEL
LIN {X 0,Y 334.551,Z 727.688,A -85,B 0,C 180,E1 13787.604,E2 13787.604} C_VEL
LIN {X 0,Y 340.215,Z 709.89,A -85,B 0,C 180,E1 13792.919,E2 13792.919} C_VEL
LIN {X 0,Y 346.554,Z 688.471,A -85,B 0,C 180,E1 13797.307,E2 13797.307} C_VEL
LIN {X 0,Y 352.947,Z 663.224,A -85,B 0,C 180,E1 13800.984,E2 13800.984} C_VEL
LIN {X 0,Y 347.725,Z 637.589,A -85,B 0,C 180,E1 13805.082,E2 13805.082} C_VEL
LIN {X 0,Y 338.339,Z 610.753,A -85,B 0,C 180,E1 13809.123,E2 13809.123} C_VEL
LIN {X 0,Y 325.215,Z 585.42,A -85,B 0,C 180,E1 13813.125,E2 13813.125} C_VEL
LIN {X 0,Y 323.557,Z 580.66,A -85,B 0,C 180,E1 13813.793,E2 13813.793} C_VEL
LIN {X 0,Y 323.503,Z 580.66,A -85,B 0,C 180,E1 13819.054,E2 13819.054} C_VEL
LIN {X 0,Y 323.624,Z 580.66,A -85,B 0,C 180,E1 13825.838,E2 13825.838} C_VEL
LIN {X 0,Y 323.95,Z 580.66,A -85,B 0,C 180,E1 13832.627,E2 13832.627} C_VEL
LIN {X 0,Y 324.3,Z 580.66,A -85,B 0,C 180,E1 13840.917,E2 13840.917} C_VEL
LIN {X 0,Y 324.672,Z 580.66,A -85,B 0,C 180,E1 13849.242,E2 13849.242} C_VEL
LIN {X 0,Y 325.436,Z 580.66,A -85,B 0,C 180,E1 13857.326,E2 13857.326} C_VEL
LIN {X 0,Y 325.364,Z 580.66,A -85,B 0,C 180,E1 13862.66,E2 13862.66} C_VEL
LIN {X 0,Y 324.755,Z 580.66,A -85,B 0,C 180,E1 13870.74,E2 13870.74} C_VEL
LIN {X 0,Y 324.327,Z 580.66,A -85,B 0,C 180,E1 13879.065,E2 13879.065} C_VEL
LIN {X 0,Y 323.964,Z 580.66,A -85,B 0,C 180,E1 13887.378,E2 13887.378} C_VEL
LIN {X 0,Y 323.657,Z 580.66,A -85,B 0,C 180,E1 13894.14,E2 13894.14} C_VEL
LIN {X 0,Y 323.66,Z 581.047,A -85,B 0,C 180,E1 13900.117,E2 13900.117} C_VEL
LIN {X 0,Y 326.442,Z 586.625,A -85,B 0,C 180,E1 13900.818,E2 13900.818} C_VEL
LIN {X 0,Y 346.181,Z 622.261,A -85,B 0,C 180,E1 13905.171,E2 13905.171} C_VEL
LIN {X 0,Y 359.393,Z 654.871,A -85,B 0,C 180,E1 13908.394,E2 13908.394} C_VEL
LIN {X 0,Y 360.554,Z 662.022,A -85,B 0,C 180,E1 13908.952,E2 13908.952} C_VEL
LIN {X 0,Y 354.623,Z 697.463,A -85,B 0,C 180,E1 13910.967,E2 13910.967} C_VEL
LIN {X 0,Y 347.584,Z 731.907,A -85,B 0,C 180,E1 13914.017,E2 13914.017} C_VEL
LIN {X 0,Y 340.301,Z 763.987,A -85,B 0,C 180,E1 13918.105,E2 13918.105} C_VEL
LIN {X 0,Y 334.048,Z 791.521,A -85,B 0,C 180,E1 13923.046,E2 13923.046} C_VEL
LIN {X 0,Y 329.46,Z 815.183,A -85,B 0,C 180,E1 13928.945,E2 13928.945} C_VEL
LIN {X 0,Y 327.308,Z 832.603,A -85,B 0,C 180,E1 13935.237,E2 13935.237} C_VEL
LIN {X 0,Y 326.923,Z 842.563,A -85,B 0,C 180,E1 13940.669,E2 13940.669} C_VEL
LIN {X 0,Y 327.097,Z 847.045,A -85,B 0,C 180,E1 13944.686,E2 13944.686} C_VEL
LIN {X 0,Y 327.253,Z 849.267,A -85,B 0,C 180,E1 13949.998,E2 13949.998} C_VEL
LIN {X 0,Y 327.046,Z 846.341,A -85,B 0,C 180,E1 13956.152,E2 13956.152} C_VEL
LIN {X 0,Y 326.981,Z 838.22,A -85,B 0,C 180,E1 13962.024,E2 13962.024} C_VEL
LIN {X 0,Y 328.145,Z 824.089,A -85,B 0,C 180,E1 13968.143,E2 13968.143} C_VEL
LIN {X 0,Y 331.414,Z 804.415,A -85,B 0,C 180,E1 13973.999,E2 13973.999} C_VEL
LIN {X 0,Y 336.933,Z 778.516,A -85,B 0,C 180,E1 13979.5,E2 13979.5} C_VEL
LIN {X 0,Y 342.742,Z 753.838,A -85,B 0,C 180,E1 13983.352,E2 13983.352} C_VEL
LIN {X 0,Y 340.996,Z 745.598,A -85,B 0,C 180,E1 13984.735,E2 13984.735} C_VEL
LIN {X 0,Y 339.288,Z 738.12,A -85,B 0,C 180,E1 13985.941,E2 13985.941} C_VEL
LIN {X 0,Y 339.513,Z 736.933,A -85,B 0,C 180,E1 13986.088,E2 13986.088} C_VEL
LIN {X 0,Y 347.252,Z 701.989,A -85,B 0,C 180,E1 13989.411,E2 13989.411} C_VEL
LIN {X 0,Y 353.554,Z 666.834,A -85,B 0,C 180,E1 13991.603,E2 13991.603} C_VEL
LIN {X 0,Y 353.808,Z 660.12,A -85,B 0,C 180,E1 13992.004,E2 13992.004} C_VEL
LIN {X 0,Y 341.027,Z 626.934,A -85,B 0,C 180,E1 13995.463,E2 13995.463} C_VEL
LIN {X 0,Y 324.152,Z 596.201,A -85,B 0,C 180,E1 13999.315,E2 13999.315} C_VEL
LIN {X 0,Y 315.9,Z 582.279,A -85,B 0,C 180,E1 14001.392,E2 14001.392} C_VEL
LIN {X 0,Y 315.721,Z 580.66,A -85,B 0,C 180,E1 14001.58,E2 14001.58} C_VEL
LIN {X 0,Y 315.79,Z 580.66,A -85,B 0,C 180,E1 14009.649,E2 14009.649} C_VEL
LIN {X 0,Y 316.151,Z 580.66,A -85,B 0,C 180,E1 14017.482,E2 14017.482} C_VEL
LIN {X 0,Y 316.455,Z 580.66,A -85,B 0,C 180,E1 14023.326,E2 14023.326} C_VEL
LIN {X 0,Y 316.985,Z 580.66,A -85,B 0,C 180,E1 14031.769,E2 14031.769} C_VEL
LIN {X 0,Y 317.666,Z 580.66,A -85,B 0,C 180,E1 14040.008,E2 14040.008} C_VEL
LIN {X 0,Y 316.976,Z 580.66,A -85,B 0,C 180,E1 14048.246,E2 14048.246} C_VEL
LIN {X 0,Y 316.51,Z 580.66,A -85,B 0,C 180,E1 14056.687,E2 14056.687} C_VEL
LIN {X 0,Y 316.08,Z 580.66,A -85,B 0,C 180,E1 14064.487,E2 14064.487} C_VEL
LIN {X 0,Y 315.8,Z 580.66,A -85,B 0,C 180,E1 14071.837,E2 14071.837} C_VEL
LIN {X 0,Y 315.511,Z 580.66,A -85,B 0,C 180,E1 14079.849,E2 14079.849} C_VEL
LIN {X 0,Y 315.573,Z 581.423,A -85,B 0,C 180,E1 14084.655,E2 14084.655} C_VEL
LIN {X 0,Y 321.688,Z 592.467,A -85,B 0,C 180,E1 14086.498,E2 14086.498} C_VEL
LIN {X 0,Y 335.022,Z 620.874,A -85,B 0,C 180,E1 14091.112,E2 14091.112} C_VEL
LIN {X 0,Y 342.817,Z 646.935,A -85,B 0,C 180,E1 14095.231,E2 14095.231} C_VEL
LIN {X 0,Y 345.999,Z 666.556,A -85,B 0,C 180,E1 14098.516,E2 14098.516} C_VEL
LIN {X 0,Y 339.008,Z 692.131,A -85,B 0,C 180,E1 14102.399,E2 14102.399} C_VEL
LIN {X 0,Y 332.2,Z 713.997,A -85,B 0,C 180,E1 14107.21,E2 14107.21} C_VEL
LIN {X 0,Y 326.48,Z 730.963,A -85,B 0,C 180,E1 14112.672,E2 14112.672} C_VEL
LIN {X 0,Y 322.772,Z 742.495,A -85,B 0,C 180,E1 14118.503,E2 14118.503} C_VEL
LIN {X 0,Y 320.906,Z 749.094,A -85,B 0,C 180,E1 14124.588,E2 14124.588} C_VEL
LIN {X 0,Y 320.335,Z 750.892,A -85,B 0,C 180,E1 14130.002,E2 14130.002} C_VEL
LIN {X 0,Y 320.91,Z 749.021,A -85,B 0,C 180,E1 14135.417,E2 14135.417} C_VEL
LIN {X 0,Y 322.804,Z 742.323,A -85,B 0,C 180,E1 14141.501,E2 14141.501} C_VEL
LIN {X 0,Y 326.559,Z 730.643,A -85,B 0,C 180,E1 14147.353,E2 14147.353} C_VEL
LIN {X 0,Y 332.227,Z 713.599,A -85,B 0,C 180,E1 14152.793,E2 14152.793} C_VEL
LIN {X 0,Y 339.19,Z 691.557,A -85,B 0,C 180,E1 14157.59,E2 14157.59} C_VEL
LIN {X 0,Y 345.946,Z 666.53,A -85,B 0,C 180,E1 14161.381,E2 14161.381} C_VEL
LIN {X 0,Y 341.8,Z 643.049,A -85,B 0,C 180,E1 14165.278,E2 14165.278} C_VEL
LIN {X 0,Y 333.291,Z 616.696,A -85,B 0,C 180,E1 14169.432,E2 14169.432} C_VEL
LIN {X 0,Y 320.787,Z 591.331,A -85,B 0,C 180,E1 14173.616,E2 14173.616} C_VEL
LIN {X 0,Y 315.6,Z 581.325,A -85,B 0,C 180,E1 14175.211,E2 14175.211} C_VEL
LIN {X 0,Y 315.53,Z 580.66,A -85,B 0,C 180,E1 14181.397,E2 14181.397} C_VEL
LIN {X 0,Y 315.769,Z 580.66,A -85,B 0,C 180,E1 14189.665,E2 14189.665} C_VEL
LIN {X 0,Y 316.171,Z 580.66,A -85,B 0,C 180,E1 14197.466,E2 14197.466} C_VEL
LIN {X 0,Y 316.454,Z 580.66,A -85,B 0,C 180,E1 14203.31,E2 14203.31} C_VEL
LIN {X 0,Y 317.002,Z 580.66,A -85,B 0,C 180,E1 14211.791,E2 14211.791} C_VEL
LIN {X 0,Y 317.679,Z 580.66,A -85,B 0,C 180,E1 14219.992,E2 14219.992} C_VEL
LIN {X 0,Y 316.991,Z 580.66,A -85,B 0,C 180,E1 14228.23,E2 14228.23} C_VEL
LIN {X 0,Y 316.521,Z 580.66,A -85,B 0,C 180,E1 14236.67,E2 14236.67} C_VEL
LIN {X 0,Y 316.08,Z 580.66,A -85,B 0,C 180,E1 14244.475,E2 14244.475} C_VEL
LIN {X 0,Y 315.769,Z 580.66,A -85,B 0,C 180,E1 14251.822,E2 14251.822} C_VEL
LIN {X 0,Y 315.719,Z 580.767,A -85,B 0,C 180,E1 14258.556,E2 14258.556} C_VEL
LIN {X 0,Y 318.076,Z 586.259,A -85,B 0,C 180,E1 14259.22,E2 14259.22} C_VEL
LIN {X 0,Y 336.504,Z 617.891,A -85,B 0,C 180,E1 14263.539,E2 14263.539} C_VEL
LIN {X 0,Y 350.689,Z 650.475,A -85,B 0,C 180,E1 14267.044,E2 14267.044} C_VEL
LIN {X 0,Y 354.098,Z 663.179,A -85,B 0,C 180,E1 14268.234,E2 14268.234} C_VEL
LIN {X 0,Y 347.576,Z 699.772,A -85,B 0,C 180,E1 14270.424,E2 14270.424} C_VEL
LIN {X 0,Y 340.469,Z 732.831,A -85,B 0,C 180,E1 14273.469,E2 14273.469} C_VEL
LIN {X 0,Y 332.829,Z 764.674,A -85,B 0,C 180,E1 14277.687,E2 14277.687} C_VEL
LIN {X 0,Y 326.359,Z 791.774,A -85,B 0,C 180,E1 14282.732,E2 14282.732} C_VEL
LIN {X 0,Y 321.736,Z 814.502,A -85,B 0,C 180,E1 14288.608,E2 14288.608} C_VEL
LIN {X 0,Y 319.482,Z 831.404,A -85,B 0,C 180,E1 14294.889,E2 14294.889} C_VEL
LIN {X 0,Y 319.092,Z 841.351,A -85,B 0,C 180,E1 14300.438,E2 14300.438} C_VEL
LIN {X 0,Y 319.28,Z 845.94,A -85,B 0,C 180,E1 14304.678,E2 14304.678} C_VEL
LIN {X 0,Y 319.438,Z 848.08,A -85,B 0,C 180,E1 14309.997,E2 14309.997} C_VEL
LIN {X 0,Y 319.262,Z 845.859,A -85,B 0,C 180,E1 14315.44,E2 14315.44} C_VEL
LIN {X 0,Y 319.091,Z 839.296,A -85,B 0,C 180,E1 14320.938,E2 14320.938} C_VEL
LIN {X 0,Y 319.946,Z 826.539,A -85,B 0,C 180,E1 14327.186,E2 14327.186} C_VEL
LIN {X 0,Y 323.114,Z 807.086,A -85,B 0,C 180,E1 14333.548,E2 14333.548} C_VEL
LIN {X 0,Y 328.547,Z 782.525,A -85,B 0,C 180,E1 14339.189,E2 14339.189} C_VEL
LIN {X 0,Y 335.763,Z 753.068,A -85,B 0,C 180,E1 14344.038,E2 14344.038} C_VEL
LIN {X 0,Y 339.513,Z 736.933,A -85,B 0,C 180,E1 14346.088,E2 14346.088} C_VEL
LIN {X 0,Y 339.451,Z 723.132,A -85,B 0,C 180,E1 14347.912,E2 14347.912} C_VEL
LIN {X 0,Y 339.301,Z 708.717,A -85,B 0,C 180,E1 14349.593,E2 14349.593} C_VEL
LIN {X 0,Y 346.222,Z 673.166,A -85,B 0,C 180,E1 14352.074,E2 14352.074} C_VEL
LIN {X 0,Y 347.404,Z 662.741,A -85,B 0,C 180,E1 14352.666,E2 14352.666} C_VEL
LIN {X 0,Y 335.018,Z 630.007,A -85,B 0,C 180,E1 14356.262,E2 14356.262} C_VEL
LIN {X 0,Y 317.877,Z 598.25,A -85,B 0,C 180,E1 14360.438,E2 14360.438} C_VEL
LIN {X 0,Y 307.893,Z 581.974,A -85,B 0,C 180,E1 14363.101,E2 14363.101} C_VEL
LIN {X 0,Y 307.764,Z 580.66,A -85,B 0,C 180,E1 14363.25,E2 14363.25} C_VEL
LIN {X 0,Y 307.894,Z 580.66,A -85,B 0,C 180,E1 14370.554,E2 14370.554} C_VEL
LIN {X 0,Y 308.238,Z 580.66,A -85,B 0,C 180,E1 14378.94,E2 14378.94} C_VEL
LIN {X 0,Y 308.613,Z 580.66,A -85,B 0,C 180,E1 14385.809,E2 14385.809} C_VEL
LIN {X 0,Y 309.272,Z 580.66,A -85,B 0,C 180,E1 14394.389,E2 14394.389} C_VEL
LIN {X 0,Y 309.763,Z 580.66,A -85,B 0,C 180,E1 14400.008,E2 14400.008} C_VEL
LIN {X 0,Y 309.314,Z 580.66,A -85,B 0,C 180,E1 14405.626,E2 14405.626} C_VEL
LIN {X 0,Y 308.693,Z 580.66,A -85,B 0,C 180,E1 14414.204,E2 14414.204} C_VEL
LIN {X 0,Y 308.262,Z 580.66,A -85,B 0,C 180,E1 14421.071,E2 14421.071} C_VEL
LIN {X 0,Y 307.926,Z 580.66,A -85,B 0,C 180,E1 14429.46,E2 14429.46} C_VEL
LIN {X 0,Y 307.596,Z 580.66,A -85,B 0,C 180,E1 14438.048,E2 14438.048} C_VEL
LIN {X 0,Y 307.569,Z 580.66,A -85,B 0,C 180,E1 14442.864,E2 14442.864} C_VEL
LIN {X 0,Y 309.932,Z 586.316,A -85,B 0,C 180,E1 14443.714,E2 14443.714} C_VEL
LIN {X 0,Y 322.524,Z 609.365,A -85,B 0,C 180,E1 14447.902,E2 14447.902} C_VEL
LIN {X 0,Y 332.253,Z 634.46,A -85,B 0,C 180,E1 14452.1,E2 14452.1} C_VEL
LIN {X 0,Y 337.846,Z 659.077,A -85,B 0,C 180,E1 14456.22,E2 14456.22} C_VEL
LIN {X 0,Y 338.895,Z 669.944,A -85,B 0,C 180,E1 14458.098,E2 14458.098} C_VEL
LIN {X 0,Y 331.581,Z 695.044,A -85,B 0,C 180,E1 14462.097,E2 14462.097} C_VEL
LIN {X 0,Y 324.578,Z 716.467,A -85,B 0,C 180,E1 14467.007,E2 14467.007} C_VEL
LIN {X 0,Y 318.527,Z 733.57,A -85,B 0,C 180,E1 14472.853,E2 14472.853} C_VEL
LIN {X 0,Y 314.836,Z 744.708,A -85,B 0,C 180,E1 14478.912,E2 14478.912} C_VEL
LIN {X 0,Y 313.147,Z 750.278,A -85,B 0,C 180,E1 14484.454,E2 14484.454} C_VEL
LIN {X 0,Y 312.525,Z 752.078,A -85,B 0,C 180,E1 14490.003,E2 14490.003} C_VEL
LIN {X 0,Y 313.151,Z 750.207,A -85,B 0,C 180,E1 14495.551,E2 14495.551} C_VEL
LIN {X 0,Y 315.497,Z 742.474,A -85,B 0,C 180,E1 14502.474,E2 14502.474} C_VEL
LIN {X 0,Y 320.021,Z 729.04,A -85,B 0,C 180,E1 14508.855,E2 14508.855} C_VEL
LIN {X 0,Y 326.337,Z 711.044,A -85,B 0,C 180,E1 14514.317,E2 14514.317} C_VEL
LIN {X 0,Y 333.328,Z 689.193,A -85,B 0,C 180,E1 14518.858,E2 14518.858} C_VEL
LIN {X 0,Y 339.071,Z 667.482,A -85,B 0,C 180,E1 14522.164,E2 14522.164} C_VEL
LIN {X 0,Y 334.6,Z 643.173,A -85,B 0,C 180,E1 14526.35,E2 14526.35} C_VEL
LIN {X 0,Y 326.254,Z 617.977,A -85,B 0,C 180,E1 14530.521,E2 14530.521} C_VEL
LIN {X 0,Y 313.473,Z 592.169,A -85,B 0,C 180,E1 14535.033,E2 14535.033} C_VEL
LIN {X 0,Y 307.638,Z 581.572,A -85,B 0,C 180,E1 14536.911,E2 14536.911} C_VEL
LIN {X 0,Y 307.576,Z 580.66,A -85,B 0,C 180,E1 14537.057,E2 14537.057} C_VEL
LIN {X 0,Y 307.59,Z 580.66,A -85,B 0,C 180,E1 14543.786,E2 14543.786} C_VEL
LIN {X 0,Y 307.92,Z 580.66,A -85,B 0,C 180,E1 14552.263,E2 14552.263} C_VEL
LIN {X 0,Y 308.362,Z 580.66,A -85,B 0,C 180,E1 14559.89,E2 14559.89} C_VEL
LIN {X 0,Y 308.586,Z 580.66,A -85,B 0,C 180,E1 14565.791,E2 14565.791} C_VEL
LIN {X 0,Y 309.304,Z 580.66,A -85,B 0,C 180,E1 14574.374,E2 14574.374} C_VEL
LIN {X 0,Y 309.775,Z 580.66,A -85,B 0,C 180,E1 14579.992,E2 14579.992} C_VEL
LIN {X 0,Y 309.05,Z 580.66,A -85,B 0,C 180,E1 14588.443,E2 14588.443} C_VEL
LIN {X 0,Y 308.576,Z 580.66,A -85,B 0,C 180,E1 14597.113,E2 14597.113} C_VEL
LIN {X 0,Y 308.203,Z 580.66,A -85,B 0,C 180,E1 14603.132,E2 14603.132} C_VEL
LIN {X 0,Y 307.906,Z 580.66,A -85,B 0,C 180,E1 14609.445,E2 14609.445} C_VEL
LIN {X 0,Y 307.805,Z 581.45,A -85,B 0,C 180,E1 14616.9,E2 14616.9} C_VEL
LIN {X 0,Y 310.562,Z 586.679,A -85,B 0,C 180,E1 14617.695,E2 14617.695} C_VEL
LIN {X 0,Y 329.32,Z 618.491,A -85,B 0,C 180,E1 14622.377,E2 14622.377} C_VEL
LIN {X 0,Y 342.993,Z 649.427,A -85,B 0,C 180,E1 14625.936,E2 14625.936} C_VEL
LIN {X 0,Y 347.47,Z 665.507,A -85,B 0,C 180,E1 14627.559,E2 14627.559} C_VEL
LIN {X 0,Y 340.959,Z 700.133,A -85,B 0,C 180,E1 14629.708,E2 14629.708} C_VEL
LIN {X 0,Y 333.329,Z 734.048,A -85,B 0,C 180,E1 14632.931,E2 14632.931} C_VEL
LIN {X 0,Y 325.485,Z 764.898,A -85,B 0,C 180,E1 14637.174,E2 14637.174} C_VEL
LIN {X 0,Y 318.697,Z 792.033,A -85,B 0,C 180,E1 14642.404,E2 14642.404} C_VEL
LIN {X 0,Y 313.923,Z 814.307,A -85,B 0,C 180,E1 14648.421,E2 14648.421} C_VEL
LIN {X 0,Y 311.704,Z 830.163,A -85,B 0,C 180,E1 14654.503,E2 14654.503} C_VEL
LIN {X 0,Y 311.257,Z 840.139,A -85,B 0,C 180,E1 14660.195,E2 14660.195} C_VEL
LIN {X 0,Y 311.425,Z 844.65,A -85,B 0,C 180,E1 14664.418,E2 14664.418} C_VEL
LIN {X 0,Y 311.631,Z 846.894,A -85,B 0,C 180,E1 14669.997,E2 14669.997} C_VEL
LIN {X 0,Y 311.423,Z 844.662,A -85,B 0,C 180,E1 14675.577,E2 14675.577} C_VEL
LIN {X 0,Y 311.253,Z 838.076,A -85,B 0,C 180,E1 14681.217,E2 14681.217} C_VEL
LIN {X 0,Y 312.189,Z 825.396,A -85,B 0,C 180,E1 14687.582,E2 14687.582} C_VEL
LIN {X 0,Y 315.463,Z 806.502,A -85,B 0,C 180,E1 14693.952,E2 14693.952} C_VEL
LIN {X 0,Y 321.025,Z 782.551,A -85,B 0,C 180,E1 14699.635,E2 14699.635} C_VEL
LIN {X 0,Y 328.524,Z 753.594,A -85,B 0,C 180,E1 14704.568,E2 14704.568} C_VEL
LIN {X 0,Y 336.401,Z 721.105,A -85,B 0,C 180,E1 14708.459,E2 14708.459} C_VEL
LIN {X 0,Y 339.301,Z 708.717,A -85,B 0,C 180,E1 14709.593,E2 14709.593} C_VEL
LIN {X 0,Y 339.184,Z 693.849,A -85,B 0,C 180,E1 14711.168,E2 14711.168} C_VEL
LIN {X 0,Y 338.687,Z 680.502,A -85,B 0,C 180,E1 14712.442,E2 14712.442} C_VEL
LIN {X 0,Y 338.977,Z 678.479,A -85,B 0,C 180,E1 14712.571,E2 14712.571} C_VEL
LIN {X 0,Y 340.965,Z 665.382,A -85,B 0,C 180,E1 14713.329,E2 14713.329} C_VEL
LIN {X 0,Y 329.317,Z 633.693,A -85,B 0,C 180,E1 14717.009,E2 14717.009} C_VEL
LIN {X 0,Y 313.491,Z 603.773,A -85,B 0,C 180,E1 14721.119,E2 14721.119} C_VEL
LIN {X 0,Y 301.98,Z 586.139,A -85,B 0,C 180,E1 14724.295,E2 14724.295} C_VEL
LIN {X 0,Y 299.735,Z 580.66,A -85,B 0,C 180,E1 14725.128,E2 14725.128} C_VEL
LIN {X 0,Y 300.06,Z 580.66,A -85,B 0,C 180,E1 14733.001,E2 14733.001} C_VEL
LIN {X 0,Y 300.378,Z 580.66,A -85,B 0,C 180,E1 14739.348,E2 14739.348} C_VEL
LIN {X 0,Y 300.652,Z 580.66,A -85,B 0,C 180,E1 14745.425,E2 14745.425} C_VEL
LIN {X 0,Y 301.345,Z 580.66,A -85,B 0,C 180,E1 14754.241,E2 14754.241} C_VEL
LIN {X 0,Y 301.869,Z 580.66,A -85,B 0,C 180,E1 14760.008,E2 14760.008} C_VEL
LIN {X 0,Y 301.381,Z 580.66,A -85,B 0,C 180,E1 14765.774,E2 14765.774} C_VEL
LIN {X 0,Y 300.729,Z 580.66,A -85,B 0,C 180,E1 14774.588,E2 14774.588} C_VEL
LIN {X 0,Y 300.405,Z 580.66,A -85,B 0,C 180,E1 14780.667,E2 14780.667} C_VEL
LIN {X 0,Y 300.082,Z 580.66,A -85,B 0,C 180,E1 14787.015,E2 14787.015} C_VEL
LIN {X 0,Y 299.753,Z 580.66,A -85,B 0,C 180,E1 14793.762,E2 14793.762} C_VEL
LIN {X 0,Y 299.684,Z 581.445,A -85,B 0,C 180,E1 14801.065,E2 14801.065} C_VEL
LIN {X 0,Y 302.503,Z 586.704,A -85,B 0,C 180,E1 14802.049,E2 14802.049} C_VEL
LIN {X 0,Y 316.163,Z 612.151,A -85,B 0,C 180,E1 14806.925,E2 14806.925} C_VEL
LIN {X 0,Y 325.693,Z 636.909,A -85,B 0,C 180,E1 14811.299,E2 14811.299} C_VEL
LIN {X 0,Y 330.949,Z 660.711,A -85,B 0,C 180,E1 14815.446,E2 14815.446} C_VEL
LIN {X 0,Y 331.857,Z 672.844,A -85,B 0,C 180,E1 14817.602,E2 14817.602} C_VEL
LIN {X 0,Y 324.189,Z 697.952,A -85,B 0,C 180,E1 14821.783,E2 14821.783} C_VEL
LIN {X 0,Y 316.958,Z 718.869,A -85,B 0,C 180,E1 14826.794,E2 14826.794} C_VEL
LIN {X 0,Y 310.968,Z 735.038,A -85,B 0,C 180,E1 14832.546,E2 14832.546} C_VEL
LIN {X 0,Y 307.153,Z 745.901,A -85,B 0,C 180,E1 14838.631,E2 14838.631} C_VEL
LIN {X 0,Y 305.383,Z 751.463,A -85,B 0,C 180,E1 14844.312,E2 14844.312} C_VEL
LIN {X 0,Y 304.716,Z 753.265,A -85,B 0,C 180,E1 14850.003,E2 14850.003} C_VEL
LIN {X 0,Y 305.386,Z 751.393,A -85,B 0,C 180,E1 14855.693,E2 14855.693} C_VEL
LIN {X 0,Y 307.875,Z 743.666,A -85,B 0,C 180,E1 14862.788,E2 14862.788} C_VEL
LIN {X 0,Y 312.641,Z 730.245,A -85,B 0,C 180,E1 14869.318,E2 14869.318} C_VEL
LIN {X 0,Y 319.233,Z 712.28,A -85,B 0,C 180,E1 14874.895,E2 14874.895} C_VEL
LIN {X 0,Y 326.524,Z 690.463,A -85,B 0,C 180,E1 14879.518,E2 14879.518} C_VEL
LIN {X 0,Y 332.22,Z 670.089,A -85,B 0,C 180,E1 14882.705,E2 14882.705} C_VEL
LIN {X 0,Y 327.824,Z 645.106,A -85,B 0,C 180,E1 14887.178,E2 14887.178} C_VEL
LIN {X 0,Y 319.585,Z 619.862,A -85,B 0,C 180,E1 14891.551,E2 14891.551} C_VEL
LIN {X 0,Y 307.362,Z 595.188,A -85,B 0,C 180,E1 14896.145,E2 14896.145} C_VEL
LIN {X 0,Y 299.716,Z 581.5,A -85,B 0,C 180,E1 14898.779,E2 14898.779} C_VEL
LIN {X 0,Y 299.659,Z 580.66,A -85,B 0,C 180,E1 14899.281,E2 14899.281} C_VEL
LIN {X 0,Y 299.699,Z 580.66,A -85,B 0,C 180,E1 14906.231,E2 14906.231} C_VEL
LIN {X 0,Y 300.068,Z 580.66,A -85,B 0,C 180,E1 14912.984,E2 14912.984} C_VEL
LIN {X 0,Y 300.401,Z 580.66,A -85,B 0,C 180,E1 14919.333,E2 14919.333} C_VEL
LIN {X 0,Y 300.63,Z 580.66,A -85,B 0,C 180,E1 14925.407,E2 14925.407} C_VEL
LIN {X 0,Y 301.376,Z 580.66,A -85,B 0,C 180,E1 14934.225,E2 14934.225} C_VEL
LIN {X 0,Y 301.884,Z 580.66,A -85,B 0,C 180,E1 14939.992,E2 14939.992} C_VEL
LIN {X 0,Y 301.122,Z 580.66,A -85,B 0,C 180,E1 14948.667,E2 14948.667} C_VEL
LIN {X 0,Y 300.669,Z 580.66,A -85,B 0,C 180,E1 14956.905,E2 14956.905} C_VEL
LIN {X 0,Y 300.114,Z 580.66,A -85,B 0,C 180,E1 14964.754,E2 14964.754} C_VEL
LIN {X 0,Y 299.811,Z 580.66,A -85,B 0,C 180,E1 14970.848,E2 14970.848} C_VEL
LIN {X 0,Y 299.735,Z 580.758,A -85,B 0,C 180,E1 14975.004,E2 14975.004} C_VEL
LIN {X 0,Y 302.018,Z 586.192,A -85,B 0,C 180,E1 14975.762,E2 14975.762} C_VEL
LIN {X 0,Y 317.367,Z 610.341,A -85,B 0,C 180,E1 14979.917,E2 14979.917} C_VEL
LIN {X 0,Y 332.601,Z 641.386,A -85,B 0,C 180,E1 14983.948,E2 14983.948} C_VEL
LIN {X 0,Y 341.036,Z 666.946,A -85,B 0,C 180,E1 14986.818,E2 14986.818} C_VEL
LIN {X 0,Y 334.405,Z 700.5,A -85,B 0,C 180,E1 14988.964,E2 14988.964} C_VEL
LIN {X 0,Y 326.36,Z 734.517,A -85,B 0,C 180,E1 14992.294,E2 14992.294} C_VEL
LIN {X 0,Y 318.381,Z 764.444,A -85,B 0,C 180,E1 14996.526,E2 14996.526} C_VEL
LIN {X 0,Y 311.393,Z 790.71,A -85,B 0,C 180,E1 15001.699,E2 15001.699} C_VEL
LIN {X 0,Y 306.382,Z 813.044,A -85,B 0,C 180,E1 15007.862,E2 15007.862} C_VEL
LIN {X 0,Y 303.912,Z 828.919,A -85,B 0,C 180,E1 15014.095,E2 15014.095} C_VEL
LIN {X 0,Y 303.387,Z 838.92,A -85,B 0,C 180,E1 15019.938,E2 15019.938} C_VEL
LIN {X 0,Y 303.526,Z 844.557,A -85,B 0,C 180,E1 15025.937,E2 15025.937} C_VEL
LIN {X 0,Y 303.815,Z 845.707,A -85,B 0,C 180,E1 15029.997,E2 15029.997} C_VEL
LIN {X 0,Y 303.569,Z 843.462,A -85,B 0,C 180,E1 15035.722,E2 15035.722} C_VEL
LIN {X 0,Y 303.397,Z 836.852,A -85,B 0,C 180,E1 15041.511,E2 15041.511} C_VEL
LIN {X 0,Y 304.545,Z 823.361,A -85,B 0,C 180,E1 15048.378,E2 15048.378} C_VEL
LIN {X 0,Y 308.247,Z 803.585,A -85,B 0,C 180,E1 15055.025,E2 15055.025} C_VEL
LIN {X 0,Y 314.461,Z 778.956,A -85,B 0,C 180,E1 15060.846,E2 15060.846} C_VEL
LIN {X 0,Y 322.382,Z 749.824,A -85,B 0,C 180,E1 15065.737,E2 15065.737} C_VEL
LIN {X 0,Y 330.289,Z 718.919,A -85,B 0,C 180,E1 15069.402,E2 15069.402} C_VEL
LIN {X 0,Y 338.114,Z 682.902,A -85,B 0,C 180,E1 15072.314,E2 15072.314} C_VEL
LIN {X 0,Y 338.977,Z 678.479,A -85,B 0,C 180,E1 15072.571,E2 15072.571} C_VEL
LIN {X 0,Y 338.18,Z 669.036,A -85,B 0,C 180,E1 15073.444,E2 15073.444} C_VEL
LIN {X 0,Y 329.096,Z 651.027,A -85,B 0,C 180,E1 15076.052,E2 15076.052} C_VEL
LIN {X 0,Y 316.15,Z 621.766,A -85,B 0,C 180,E1 15079.911,E2 15079.911} C_VEL
LIN {X 0,Y 299.317,Z 593.359,A -85,B 0,C 180,E1 15084.645,E2 15084.645} C_VEL
LIN {X 0,Y 292.008,Z 582.473,A -85,B 0,C 180,E1 15086.952,E2 15086.952} C_VEL
LIN {X 0,Y 291.795,Z 580.66,A -85,B 0,C 180,E1 15087.165,E2 15087.165} C_VEL
LIN {X 0,Y 292.213,Z 580.66,A -85,B 0,C 180,E1 15095.521,E2 15095.521} C_VEL
LIN {X 0,Y 292.545,Z 580.66,A -85,B 0,C 180,E1 15101.918,E2 15101.918} C_VEL
LIN {X 0,Y 292.975,Z 580.66,A -85,B 0,C 180,E1 15109.059,E2 15109.059} C_VEL
LIN {X 0,Y 293.742,Z 580.66,A -85,B 0,C 180,E1 15117.054,E2 15117.054} C_VEL
LIN {X 0,Y 293.753,Z 580.66,A -85,B 0,C 180,E1 15122.963,E2 15122.963} C_VEL
LIN {X 0,Y 292.999,Z 580.66,A -85,B 0,C 180,E1 15131.937,E2 15131.937} C_VEL
LIN {X 0,Y 292.588,Z 580.66,A -85,B 0,C 180,E1 15138.097,E2 15138.097} C_VEL
LIN {X 0,Y 292.228,Z 580.66,A -85,B 0,C 180,E1 15144.496,E2 15144.496} C_VEL
LIN {X 0,Y 291.907,Z 580.66,A -85,B 0,C 180,E1 15151.253,E2 15151.253} C_VEL
LIN {X 0,Y 291.673,Z 581.017,A -85,B 0,C 180,E1 15158.961,E2 15158.961} C_VEL
LIN {X 0,Y 294.02,Z 586.278,A -85,B 0,C 180,E1 15159.909,E2 15159.909} C_VEL
LIN {X 0,Y 306.581,Z 607.914,A -85,B 0,C 180,E1 15164.54,E2 15164.54} C_VEL
LIN {X 0,Y 317.444,Z 633.64,A -85,B 0,C 180,E1 15169.422,E2 15169.422} C_VEL
LIN {X 0,Y 323.685,Z 659.21,A -85,B 0,C 180,E1 15174.06,E2 15174.06} C_VEL
LIN {X 0,Y 325.094,Z 674.873,A -85,B 0,C 180,E1 15176.974,E2 15176.974} C_VEL
LIN {X 0,Y 316.764,Z 700.868,A -85,B 0,C 180,E1 15181.45,E2 15181.45} C_VEL
LIN {X 0,Y 309.321,Z 721.211,A -85,B 0,C 180,E1 15186.569,E2 15186.569} C_VEL
LIN {X 0,Y 303.132,Z 737.274,A -85,B 0,C 180,E1 15192.565,E2 15192.565} C_VEL
LIN {X 0,Y 299.496,Z 747.089,A -85,B 0,C 180,E1 15198.337,E2 15198.337} C_VEL
LIN {X 0,Y 297.607,Z 752.649,A -85,B 0,C 180,E1 15204.163,E2 15204.163} C_VEL
LIN {X 0,Y 296.918,Z 754.449,A -85,B 0,C 180,E1 15210.003,E2 15210.003} C_VEL
LIN {X 0,Y 297.61,Z 752.582,A -85,B 0,C 180,E1 15215.842,E2 15215.842} C_VEL
LIN {X 0,Y 300.271,Z 744.856,A -85,B 0,C 180,E1 15223.117,E2 15223.117} C_VEL
LIN {X 0,Y 304.985,Z 732.174,A -85,B 0,C 180,E1 15229.522,E2 15229.522} C_VEL
LIN {X 0,Y 311.699,Z 714.784,A -85,B 0,C 180,E1 15235.154,E2 15235.154} C_VEL
LIN {X 0,Y 319.77,Z 691.733,A -85,B 0,C 180,E1 15240.206,E2 15240.206} C_VEL
LIN {X 0,Y 325.438,Z 672.846,A -85,B 0,C 180,E1 15243.236,E2 15243.236} C_VEL
LIN {X 0,Y 321.25,Z 647.58,A -85,B 0,C 180,E1 15247.946,E2 15247.946} C_VEL
LIN {X 0,Y 313.538,Z 623.231,A -85,B 0,C 180,E1 15252.369,E2 15252.369} C_VEL
LIN {X 0,Y 301.649,Z 598.544,A -85,B 0,C 180,E1 15257.211,E2 15257.211} C_VEL
LIN {X 0,Y 293.703,Z 585.928,A -85,B 0,C 180,E1 15260.046,E2 15260.046} C_VEL
LIN {X 0,Y 291.64,Z 580.66,A -85,B 0,C 180,E1 15261.147,E2 15261.147} C_VEL
LIN {X 0,Y 291.859,Z 580.66,A -85,B 0,C 180,E1 15268.742,E2 15268.742} C_VEL
LIN {X 0,Y 292.233,Z 580.66,A -85,B 0,C 180,E1 15275.505,E2 15275.505} C_VEL
LIN {X 0,Y 292.557,Z 580.66,A -85,B 0,C 180,E1 15281.901,E2 15281.901} C_VEL
LIN {X 0,Y 292.934,Z 580.66,A -85,B 0,C 180,E1 15289.13,E2 15289.13} C_VEL
LIN {X 0,Y 293.774,Z 580.66,A -85,B 0,C 180,E1 15297.038,E2 15297.038} C_VEL
LIN {X 0,Y 293.737,Z 580.66,A -85,B 0,C 180,E1 15302.946,E2 15302.946} C_VEL
LIN {X 0,Y 293.015,Z 580.66,A -85,B 0,C 180,E1 15311.92,E2 15311.92} C_VEL
LIN {X 0,Y 292.597,Z 580.66,A -85,B 0,C 180,E1 15318.079,E2 15318.079} C_VEL
LIN {X 0,Y 292.228,Z 580.66,A -85,B 0,C 180,E1 15324.477,E2 15324.477} C_VEL
LIN {X 0,Y 291.807,Z 581.056,A -85,B 0,C 180,E1 15332.985,E2 15332.985} C_VEL
LIN {X 0,Y 294.215,Z 586.31,A -85,B 0,C 180,E1 15333.845,E2 15333.845} C_VEL
LIN {X 0,Y 308.102,Z 607.659,A -85,B 0,C 180,E1 15337.941,E2 15337.941} C_VEL
LIN {X 0,Y 323.24,Z 636.323,A -85,B 0,C 180,E1 15342.123,E2 15342.123} C_VEL
LIN {X 0,Y 334.365,Z 667.568,A -85,B 0,C 180,E1 15345.943,E2 15345.943} C_VEL
LIN {X 0,Y 326.976,Z 704.973,A -85,B 0,C 180,E1 15348.536,E2 15348.536} C_VEL
LIN {X 0,Y 318.52,Z 738.296,A -85,B 0,C 180,E1 15352.048,E2 15352.048} C_VEL
LIN {X 0,Y 309.857,Z 769.118,A -85,B 0,C 180,E1 15356.746,E2 15356.746} C_VEL
LIN {X 0,Y 302.61,Z 795.3,A -85,B 0,C 180,E1 15362.429,E2 15362.429} C_VEL
LIN {X 0,Y 297.876,Z 816.072,A -85,B 0,C 180,E1 15368.765,E2 15368.765} C_VEL
LIN {X 0,Y 295.811,Z 830.646,A -85,B 0,C 180,E1 15375.17,E2 15375.17} C_VEL
LIN {X 0,Y 295.59,Z 839.522,A -85,B 0,C 180,E1 15381.158,E2 15381.158} C_VEL
LIN {X 0,Y 295.804,Z 843.89,A -85,B 0,C 180,E1 15387.063,E2 15387.063} C_VEL
LIN {X 0,Y 296.013,Z 844.522,A -85,B 0,C 180,E1 15389.997,E2 15389.997} C_VEL
LIN {X 0,Y 295.728,Z 842.264,A -85,B 0,C 180,E1 15395.874,E2 15395.874} C_VEL
LIN {X 0,Y 295.551,Z 835.629,A -85,B 0,C 180,E1 15401.821,E2 15401.821} C_VEL
LIN {X 0,Y 296.797,Z 822.328,A -85,B 0,C 180,E1 15408.778,E2 15408.778} C_VEL
LIN {X 0,Y 300.604,Z 803.189,A -85,B 0,C 180,E1 15415.435,E2 15415.435} C_VEL
LIN {X 0,Y 306.829,Z 779.7,A -85,B 0,C 180,E1 15421.203,E2 15421.203} C_VEL
LIN {X 0,Y 315.114,Z 750.845,A -85,B 0,C 180,E1 15426.266,E2 15426.266} C_VEL
LIN {X 0,Y 323.718,Z 718.782,A -85,B 0,C 180,E1 15430.18,E2 15430.18} C_VEL
LIN {X 0,Y 331.74,Z 683.44,A -85,B 0,C 180,E1 15433.106,E2 15433.106} C_VEL
LIN {X 0,Y 334.454,Z 667.545,A -85,B 0,C 180,E1 15434.071,E2 15434.071} C_VEL
LIN {X 0,Y 329.096,Z 651.027,A -85,B 0,C 180,E1 15436.052,E2 15436.052} C_VEL
LIN {X 0,Y 323.556,Z 642.525,A -85,B 0,C 180,E1 15437.517,E2 15437.517} C_VEL
LIN {X 0,Y 313.676,Z 631.362,A -85,B 0,C 180,E1 15439.909,E2 15439.909} C_VEL
LIN {X 0,Y 312.896,Z 629.741,A -85,B 0,C 180,E1 15440.145,E2 15440.145} C_VEL
LIN {X 0,Y 297.373,Z 602.569,A -85,B 0,C 180,E1 15444.748,E2 15444.748} C_VEL
LIN {X 0,Y 286.47,Z 586.45,A -85,B 0,C 180,E1 15448.32,E2 15448.32} C_VEL
LIN {X 0,Y 284.055,Z 581.793,A -85,B 0,C 180,E1 15449.244,E2 15449.244} C_VEL
LIN {X 0,Y 283.955,Z 580.66,A -85,B 0,C 180,E1 15449.577,E2 15449.577} C_VEL
LIN {X 0,Y 284.371,Z 580.66,A -85,B 0,C 180,E1 15458.128,E2 15458.128} C_VEL
LIN {X 0,Y 284.756,Z 580.66,A -85,B 0,C 180,E1 15464.592,E2 15464.592} C_VEL
LIN {X 0,Y 285.207,Z 580.66,A -85,B 0,C 180,E1 15470.845,E2 15470.845} C_VEL
LIN {X 0,Y 285.834,Z 580.66,A -85,B 0,C 180,E1 15476.972,E2 15476.972} C_VEL
LIN {X 0,Y 285.845,Z 580.66,A -85,B 0,C 180,E1 15483.045,E2 15483.045} C_VEL
LIN {X 0,Y 285.033,Z 580.66,A -85,B 0,C 180,E1 15492.276,E2 15492.276} C_VEL
LIN {X 0,Y 284.623,Z 580.66,A -85,B 0,C 180,E1 15498.621,E2 15498.621} C_VEL
LIN {X 0,Y 284.204,Z 580.66,A -85,B 0,C 180,E1 15505.235,E2 15505.235} C_VEL
LIN {X 0,Y 283.939,Z 580.66,A -85,B 0,C 180,E1 15512.234,E2 15512.234} C_VEL
LIN {X 0,Y 283.678,Z 580.66,A -85,B 0,C 180,E1 15516.618,E2 15516.618} C_VEL
LIN {X 0,Y 285.77,Z 585.992,A -85,B 0,C 180,E1 15517.596,E2 15517.596} C_VEL
LIN {X 0,Y 288.361,Z 589.631,A -85,B 0,C 180,E1 15518.581,E2 15518.581} C_VEL
LIN {X 0,Y 300.581,Z 610.807,A -85,B 0,C 180,E1 15523.456,E2 15523.456} C_VEL
LIN {X 0,Y 310.807,Z 635.538,A -85,B 0,C 180,E1 15528.392,E2 15528.392} C_VEL
LIN {X 0,Y 316.818,Z 660.287,A -85,B 0,C 180,E1 15533.086,E2 15533.086} C_VEL
LIN {X 0,Y 318.611,Z 676.166,A -85,B 0,C 180,E1 15536.213,E2 15536.213} C_VEL
LIN {X 0,Y 309.929,Z 702.117,A -85,B 0,C 180,E1 15540.761,E2 15540.761} C_VEL
LIN {X 0,Y 301.695,Z 723.552,A -85,B 0,C 180,E1 15546.333,E2 15546.333} C_VEL
LIN {X 0,Y 295.086,Z 739.916,A -85,B 0,C 180,E1 15552.844,E2 15552.844} C_VEL
LIN {X 0,Y 291.19,Z 750.022,A -85,B 0,C 180,E1 15559.518,E2 15559.518} C_VEL
LIN {X 0,Y 289.847,Z 753.834,A -85,B 0,C 180,E1 15564.006,E2 15564.006} C_VEL
LIN {X 0,Y 289.109,Z 755.636,A -85,B 0,C 180,E1 15570.003,E2 15570.003} C_VEL
LIN {X 0,Y 289.85,Z 753.768,A -85,B 0,C 180,E1 15575.999,E2 15575.999} C_VEL
LIN {X 0,Y 292.656,Z 746.049,A -85,B 0,C 180,E1 15583.465,E2 15583.465} C_VEL
LIN {X 0,Y 297.881,Z 732.791,A -85,B 0,C 180,E1 15590.259,E2 15590.259} C_VEL
LIN {X 0,Y 305.142,Z 714.743,A -85,B 0,C 180,E1 15596.129,E2 15596.129} C_VEL
LIN {X 0,Y 313.058,Z 692.998,A -85,B 0,C 180,E1 15600.923,E2 15600.923} C_VEL
LIN {X 0,Y 318.499,Z 673.852,A -85,B 0,C 180,E1 15604.134,E2 15604.134} C_VEL
LIN {X 0,Y 314.534,Z 649.246,A -85,B 0,C 180,E1 15608.895,E2 15608.895} C_VEL
LIN {X 0,Y 306.792,Z 624.785,A -85,B 0,C 180,E1 15613.572,E2 15613.572} C_VEL
LIN {X 0,Y 294.494,Z 599.186,A -85,B 0,C 180,E1 15618.91,E2 15618.91} C_VEL
LIN {X 0,Y 285.897,Z 586.128,A -85,B 0,C 180,E1 15622.2,E2 15622.2} C_VEL
LIN {X 0,Y 283.707,Z 581.559,A -85,B 0,C 180,E1 15623.138,E2 15623.138} C_VEL
LIN {X 0,Y 283.695,Z 580.66,A -85,B 0,C 180,E1 15624.042,E2 15624.042} C_VEL
LIN {X 0,Y 284.001,Z 580.66,A -85,B 0,C 180,E1 15631.318,E2 15631.318} C_VEL
LIN {X 0,Y 284.39,Z 580.66,A -85,B 0,C 180,E1 15638.111,E2 15638.111} C_VEL
LIN {X 0,Y 284.744,Z 580.66,A -85,B 0,C 180,E1 15644.573,E2 15644.573} C_VEL
LIN {X 0,Y 285.494,Z 580.66,A -85,B 0,C 180,E1 15653.903,E2 15653.903} C_VEL
LIN {X 0,Y 286.077,Z 580.66,A -85,B 0,C 180,E1 15659.992,E2 15659.992} C_VEL
LIN {X 0,Y 285.505,Z 580.66,A -85,B 0,C 180,E1 15666.08,E2 15666.08} C_VEL
LIN {X 0,Y 285.048,Z 580.66,A -85,B 0,C 180,E1 15672.258,E2 15672.258} C_VEL
LIN {X 0,Y 284.628,Z 580.66,A -85,B 0,C 180,E1 15678.603,E2 15678.603} C_VEL
LIN {X 0,Y 284.197,Z 580.66,A -85,B 0,C 180,E1 15685.217,E2 15685.217} C_VEL
LIN {X 0,Y 283.968,Z 581.101,A -85,B 0,C 180,E1 15690.763,E2 15690.763} C_VEL
LIN {X 0,Y 286.57,Z 586.54,A -85,B 0,C 180,E1 15691.774,E2 15691.774} C_VEL
LIN {X 0,Y 300.84,Z 608.115,A -85,B 0,C 180,E1 15696.344,E2 15696.344} C_VEL
LIN {X 0,Y 315.546,Z 635.504,A -85,B 0,C 180,E1 15700.701,E2 15700.701} C_VEL
LIN {X 0,Y 326.639,Z 665.363,A -85,B 0,C 180,E1 15704.639,E2 15704.639} C_VEL
LIN {X 0,Y 327.955,Z 671.893,A -85,B 0,C 180,E1 15705.362,E2 15705.362} C_VEL
LIN {X 0,Y 320.004,Z 707.297,A -85,B 0,C 180,E1 15707.925,E2 15707.925} C_VEL
LIN {X 0,Y 311.006,Z 740.828,A -85,B 0,C 180,E1 15711.63,E2 15711.63} C_VEL
LIN {X 0,Y 301.982,Z 771.097,A -85,B 0,C 180,E1 15716.527,E2 15716.527} C_VEL
LIN {X 0,Y 294.574,Z 796.866,A -85,B 0,C 180,E1 15722.444,E2 15722.444} C_VEL
LIN {X 0,Y 289.692,Z 817.098,A -85,B 0,C 180,E1 15729.084,E2 15729.084} C_VEL
LIN {X 0,Y 287.886,Z 830.673,A -85,B 0,C 180,E1 15735.501,E2 15735.501} C_VEL
LIN {X 0,Y 287.781,Z 839.79,A -85,B 0,C 180,E1 15742.439,E2 15742.439} C_VEL
LIN {X 0,Y 287.998,Z 842.739,A -85,B 0,C 180,E1 15747.077,E2 15747.077} C_VEL
LIN {X 0,Y 288.196,Z 843.334,A -85,B 0,C 180,E1 15749.997,E2 15749.997} C_VEL
LIN {X 0,Y 287.871,Z 841.063,A -85,B 0,C 180,E1 15756.035,E2 15756.035} C_VEL
LIN {X 0,Y 287.688,Z 834.403,A -85,B 0,C 180,E1 15762.149,E2 15762.149} C_VEL
LIN {X 0,Y 288.973,Z 821.859,A -85,B 0,C 180,E1 15768.946,E2 15768.946} C_VEL
LIN {X 0,Y 292.653,Z 804.064,A -85,B 0,C 180,E1 15775.475,E2 15775.475} C_VEL
LIN {X 0,Y 299.332,Z 780.102,A -85,B 0,C 180,E1 15781.649,E2 15781.649} C_VEL
LIN {X 0,Y 307.864,Z 751.713,A -85,B 0,C 180,E1 15786.821,E2 15786.821} C_VEL
LIN {X 0,Y 316.847,Z 719.955,A -85,B 0,C 180,E1 15790.861,E2 15790.861} C_VEL
LIN {X 0,Y 325.231,Z 684.956,A -85,B 0,C 180,E1 15793.855,E2 15793.855} C_VEL
LIN {X 0,Y 327.856,Z 669.431,A -85,B 0,C 180,E1 15794.885,E2 15794.885} C_VEL
LIN {X 0,Y 316.578,Z 637.697,A -85,B 0,C 180,E1 15799.007,E2 15799.007} C_VEL
LIN {X 0,Y 312.896,Z 629.741,A -85,B 0,C 180,E1 15800.145,E2 15800.145} C_VEL
LIN {X 0,Y 306.826,Z 622.186,A -85,B 0,C 180,E1 15801.774,E2 15801.774} C_VEL
LIN {X 0,Y 296.497,Z 613.003,A -85,B 0,C 180,E1 15804.52,E2 15804.52} C_VEL
LIN {X 0,Y 295.643,Z 611.54,A -85,B 0,C 180,E1 15804.797,E2 15804.797} C_VEL
LIN {X 0,Y 279.295,Z 587.038,A -85,B 0,C 180,E1 15810.471,E2 15810.471} C_VEL
LIN {X 0,Y 276.171,Z 581.79,A -85,B 0,C 180,E1 15811.768,E2 15811.768} C_VEL
LIN {X 0,Y 276.076,Z 580.66,A -85,B 0,C 180,E1 15812.078,E2 15812.078} C_VEL
LIN {X 0,Y 276.578,Z 580.66,A -85,B 0,C 180,E1 15820.835,E2 15820.835} C_VEL
LIN {X 0,Y 277.116,Z 580.66,A -85,B 0,C 180,E1 15829.538,E2 15829.538} C_VEL
LIN {X 0,Y 277.904,Z 580.66,A -85,B 0,C 180,E1 15836.886,E2 15836.886} C_VEL
LIN {X 0,Y 277.916,Z 580.66,A -85,B 0,C 180,E1 15843.132,E2 15843.132} C_VEL
LIN {X 0,Y 277.066,Z 580.66,A -85,B 0,C 180,E1 15852.635,E2 15852.635} C_VEL
LIN {X 0,Y 276.478,Z 580.66,A -85,B 0,C 180,E1 15861.427,E2 15861.427} C_VEL
LIN {X 0,Y 276.073,Z 580.66,A -85,B 0,C 180,E1 15869.586,E2 15869.586} C_VEL
LIN {X 0,Y 275.792,Z 580.696,A -85,B 0,C 180,E1 15874.091,E2 15874.091} C_VEL
LIN {X 0,Y 277.772,Z 585.894,A -85,B 0,C 180,E1 15875.081,E2 15875.081} C_VEL
LIN {X 0,Y 280.554,Z 589.623,A -85,B 0,C 180,E1 15876.254,E2 15876.254} C_VEL
LIN {X 0,Y 291.353,Z 607.728,A -85,B 0,C 180,E1 15880.888,E2 15880.888} C_VEL
LIN {X 0,Y 301.849,Z 630.786,A -85,B 0,C 180,E1 15885.949,E2 15885.949} C_VEL
LIN {X 0,Y 308.657,Z 653.996,A -85,B 0,C 180,E1 15890.607,E2 15890.607} C_VEL
LIN {X 0,Y 311.848,Z 677.499,A -85,B 0,C 180,E1 15895.371,E2 15895.371} C_VEL
LIN {X 0,Y 303.166,Z 703.361,A -85,B 0,C 180,E1 15900.043,E2 15900.043} C_VEL
LIN {X 0,Y 294.568,Z 724.762,A -85,B 0,C 180,E1 15905.724,E2 15905.724} C_VEL
LIN {X 0,Y 287.605,Z 741.114,A -85,B 0,C 180,E1 15912.383,E2 15912.383} C_VEL
LIN {X 0,Y 283.513,Z 751.211,A -85,B 0,C 180,E1 15919.231,E2 15919.231} C_VEL
LIN {X 0,Y 282.099,Z 755.017,A -85,B 0,C 180,E1 15923.841,E2 15923.841} C_VEL
LIN {X 0,Y 281.314,Z 756.82,A -85,B 0,C 180,E1 15930.003,E2 15930.003} C_VEL
LIN {X 0,Y 282.101,Z 754.952,A -85,B 0,C 180,E1 15936.165,E2 15936.165} C_VEL
LIN {X 0,Y 285.049,Z 747.243,A -85,B 0,C 180,E1 15943.831,E2 15943.831} C_VEL
LIN {X 0,Y 290.561,Z 733.996,A -85,B 0,C 180,E1 15950.792,E2 15950.792} C_VEL
LIN {X 0,Y 298.154,Z 715.97,A -85,B 0,C 180,E1 15956.79,E2 15956.79} C_VEL
LIN {X 0,Y 306.393,Z 694.268,A -85,B 0,C 180,E1 15961.673,E2 15961.673} C_VEL
LIN {X 0,Y 311.746,Z 676.578,A -85,B 0,C 180,E1 15964.709,E2 15964.709} C_VEL
LIN {X 0,Y 308.14,Z 651.857,A -85,B 0,C 180,E1 15969.702,E2 15969.702} C_VEL
LIN {X 0,Y 300.251,Z 626.718,A -85,B 0,C 180,E1 15974.772,E2 15974.772} C_VEL
LIN {X 0,Y 288.89,Z 603.195,A -85,B 0,C 180,E1 15980.048,E2 15980.048} C_VEL
LIN {X 0,Y 278.661,Z 586.742,A -85,B 0,C 180,E1 15984.394,E2 15984.394} C_VEL
LIN {X 0,Y 275.836,Z 581.841,A -85,B 0,C 180,E1 15985.655,E2 15985.655} C_VEL
LIN {X 0,Y 275.778,Z 580.66,A -85,B 0,C 180,E1 15986.136,E2 15986.136} C_VEL
LIN {X 0,Y 276.173,Z 580.66,A -85,B 0,C 180,E1 15993.977,E2 15993.977} C_VEL
LIN {X 0,Y 276.581,Z 580.66,A -85,B 0,C 180,E1 16000.816,E2 16000.816} C_VEL
LIN {X 0,Y 277.105,Z 580.66,A -85,B 0,C 180,E1 16009.582,E2 16009.582} C_VEL
LIN {X 0,Y 277.935,Z 580.66,A -85,B 0,C 180,E1 16016.869,E2 16016.869} C_VEL
LIN {X 0,Y 277.906,Z 580.66,A -85,B 0,C 180,E1 16023.114,E2 16023.114} C_VEL
LIN {X 0,Y 277.08,Z 580.66,A -85,B 0,C 180,E1 16032.616,E2 16032.616} C_VEL
LIN {X 0,Y 276.478,Z 580.66,A -85,B 0,C 180,E1 16041.411,E2 16041.411} C_VEL
LIN {X 0,Y 276.111,Z 580.781,A -85,B 0,C 180,E1 16048.233,E2 16048.233} C_VEL
LIN {X 0,Y 278.451,Z 586.285,A -85,B 0,C 180,E1 16049.288,E2 16049.288} C_VEL
LIN {X 0,Y 281.333,Z 590.124,A -85,B 0,C 180,E1 16050.386,E2 16050.386} C_VEL
LIN {X 0,Y 296.585,Z 613.472,A -85,B 0,C 180,E1 16055.574,E2 16055.574} C_VEL
LIN {X 0,Y 310.372,Z 640.216,A -85,B 0,C 180,E1 16060.028,E2 16060.028} C_VEL
LIN {X 0,Y 320.699,Z 669.266,A -85,B 0,C 180,E1 16064.032,E2 16064.032} C_VEL
LIN {X 0,Y 321.357,Z 674.518,A -85,B 0,C 180,E1 16064.615,E2 16064.615} C_VEL
LIN {X 0,Y 313.217,Z 709.092,A -85,B 0,C 180,E1 16067.239,E2 16067.239} C_VEL
LIN {X 0,Y 303.896,Z 741.872,A -85,B 0,C 180,E1 16071.022,E2 16071.022} C_VEL
LIN {X 0,Y 294.569,Z 771.632,A -85,B 0,C 180,E1 16076.013,E2 16076.013} C_VEL
LIN {X 0,Y 286.919,Z 796.899,A -85,B 0,C 180,E1 16082.072,E2 16082.072} C_VEL
LIN {X 0,Y 281.84,Z 816.921,A -85,B 0,C 180,E1 16088.936,E2 16088.936} C_VEL
LIN {X 0,Y 279.996,Z 830.446,A -85,B 0,C 180,E1 16095.697,E2 16095.697} C_VEL
LIN {X 0,Y 279.918,Z 838.582,A -85,B 0,C 180,E1 16102.226,E2 16102.226} C_VEL
LIN {X 0,Y 280.137,Z 841.506,A -85,B 0,C 180,E1 16106.899,E2 16106.899} C_VEL
LIN {X 0,Y 280.391,Z 842.149,A -85,B 0,C 180,E1 16109.997,E2 16109.997} C_VEL
LIN {X 0,Y 280.03,Z 839.865,A -85,B 0,C 180,E1 16116.205,E2 16116.205} C_VEL
LIN {X 0,Y 279.867,Z 833.182,A -85,B 0,C 180,E1 16122.494,E2 16122.494} C_VEL
LIN {X 0,Y 281.254,Z 820.604,A -85,B 0,C 180,E1 16129.487,E2 16129.487} C_VEL
LIN {X 0,Y 285.629,Z 801.439,A -85,B 0,C 180,E1 16136.606,E2 16136.606} C_VEL
LIN {X 0,Y 292.894,Z 777.069,A -85,B 0,C 180,E1 16142.869,E2 16142.869} C_VEL
LIN {X 0,Y 302.025,Z 748.085,A -85,B 0,C 180,E1 16148.109,E2 16148.109} C_VEL
LIN {X 0,Y 311.139,Z 717.019,A -85,B 0,C 180,E1 16151.993,E2 16151.993} C_VEL
LIN {X 0,Y 319.584,Z 682.711,A -85,B 0,C 180,E1 16154.903,E2 16154.903} C_VEL
LIN {X 0,Y 321.446,Z 671.969,A -85,B 0,C 180,E1 16155.635,E2 16155.635} C_VEL
LIN {X 0,Y 311.164,Z 641.825,A -85,B 0,C 180,E1 16159.753,E2 16159.753} C_VEL
LIN {X 0,Y 297.205,Z 614.428,A -85,B 0,C 180,E1 16164.283,E2 16164.283} C_VEL
LIN {X 0,Y 295.643,Z 611.54,A -85,B 0,C 180,E1 16164.797,E2 16164.797} C_VEL
LIN {X 0,Y 291.138,Z 608.056,A -85,B 0,C 180,E1 16166.103,E2 16166.103} C_VEL
LIN {X 0,Y 283.716,Z 604.925,A -85,B 0,C 180,E1 16168.28,E2 16168.28} C_VEL
LIN {X 0,Y 283.106,Z 604.082,A -85,B 0,C 180,E1 16168.496,E2 16168.496} C_VEL
LIN {X 0,Y 274.903,Z 592.198,A -85,B 0,C 180,E1 16171.668,E2 16171.668} C_VEL
LIN {X 0,Y 271.517,Z 587.091,A -85,B 0,C 180,E1 16173.136,E2 16173.136} C_VEL
LIN {X 0,Y 268.392,Z 582.218,A -85,B 0,C 180,E1 16174.59,E2 16174.59} C_VEL
LIN {X 0,Y 268.249,Z 580.66,A -85,B 0,C 180,E1 16174.958,E2 16174.958} C_VEL
LIN {X 0,Y 268.807,Z 580.66,A -85,B 0,C 180,E1 16183.653,E2 16183.653} C_VEL
LIN {X 0,Y 269.318,Z 580.66,A -85,B 0,C 180,E1 16190.3,E2 16190.3} C_VEL
LIN {X 0,Y 269.98,Z 580.66,A -85,B 0,C 180,E1 16196.794,E2 16196.794} C_VEL
LIN {X 0,Y 269.992,Z 580.66,A -85,B 0,C 180,E1 16203.224,E2 16203.224} C_VEL
LIN {X 0,Y 269.341,Z 580.66,A -85,B 0,C 180,E1 16209.718,E2 16209.718} C_VEL
LIN {X 0,Y 268.802,Z 580.66,A -85,B 0,C 180,E1 16216.771,E2 16216.771} C_VEL
LIN {X 0,Y 268.267,Z 580.66,A -85,B 0,C 180,E1 16225.453,E2 16225.453} C_VEL
LIN {X 0,Y 267.943,Z 580.66,A -85,B 0,C 180,E1 16231.161,E2 16231.161} C_VEL
LIN {X 0,Y 269.904,Z 585.919,A -85,B 0,C 180,E1 16232.271,E2 16232.271} C_VEL
LIN {X 0,Y 272.733,Z 589.282,A -85,B 0,C 180,E1 16233.592,E2 16233.592} C_VEL
LIN {X 0,Y 284.641,Z 609.056,A -85,B 0,C 180,E1 16239.182,E2 16239.182} C_VEL
LIN {X 0,Y 295.295,Z 632.648,A -85,B 0,C 180,E1 16244.71,E2 16244.71} C_VEL
LIN {X 0,Y 301.979,Z 655.348,A -85,B 0,C 180,E1 16249.526,E2 16249.526} C_VEL
LIN {X 0,Y 304.917,Z 677.574,A -85,B 0,C 180,E1 16254.184,E2 16254.184} C_VEL
LIN {X 0,Y 304.075,Z 683.91,A -85,B 0,C 180,E1 16255.379,E2 16255.379} C_VEL
LIN {X 0,Y 295.05,Z 707.97,A -85,B 0,C 180,E1 16260.067,E2 16260.067} C_VEL
LIN {X 0,Y 286.506,Z 728.195,A -85,B 0,C 180,E1 16265.827,E2 16265.827} C_VEL
LIN {X 0,Y 279.548,Z 743.719,A -85,B 0,C 180,E1 16272.673,E2 16272.673} C_VEL
LIN {X 0,Y 275.843,Z 752.4,A -85,B 0,C 180,E1 16278.927,E2 16278.927} C_VEL
LIN {X 0,Y 274.341,Z 756.202,A -85,B 0,C 180,E1 16283.666,E2 16283.666} C_VEL
LIN {X 0,Y 273.504,Z 758.006,A -85,B 0,C 180,E1 16290.003,E2 16290.003} C_VEL
LIN {X 0,Y 274.394,Z 755.962,A -85,B 0,C 180,E1 16296.615,E2 16296.615} C_VEL
LIN {X 0,Y 277.453,Z 748.435,A -85,B 0,C 180,E1 16304.218,E2 16304.218} C_VEL
LIN {X 0,Y 282.945,Z 735.914,A -85,B 0,C 180,E1 16311.055,E2 16311.055} C_VEL
LIN {X 0,Y 290.651,Z 718.449,A -85,B 0,C 180,E1 16317.119,E2 16317.119} C_VEL
LIN {X 0,Y 299.79,Z 695.534,A -85,B 0,C 180,E1 16322.455,E2 16322.455} C_VEL
LIN {X 0,Y 305.026,Z 679.711,A -85,B 0,C 180,E1 16325.215,E2 16325.215} C_VEL
LIN {X 0,Y 302.072,Z 656.313,A -85,B 0,C 180,E1 16330.158,E2 16330.158} C_VEL
LIN {X 0,Y 295.389,Z 632.94,A -85,B 0,C 180,E1 16335.085,E2 16335.085} C_VEL
LIN {X 0,Y 285.185,Z 609.994,A -85,B 0,C 180,E1 16340.415,E2 16340.415} C_VEL
LIN {X 0,Y 274.842,Z 592.928,A -85,B 0,C 180,E1 16345.212,E2 16345.212} C_VEL
LIN {X 0,Y 271.008,Z 586.96,A -85,B 0,C 180,E1 16347.046,E2 16347.046} C_VEL
LIN {X 0,Y 267.994,Z 581.998,A -85,B 0,C 180,E1 16348.534,E2 16348.534} C_VEL
LIN {X 0,Y 267.9,Z 580.66,A -85,B 0,C 180,E1 16348.766,E2 16348.766} C_VEL
LIN {X 0,Y 268.375,Z 580.66,A -85,B 0,C 180,E1 16356.73,E2 16356.73} C_VEL
LIN {X 0,Y 268.806,Z 580.66,A -85,B 0,C 180,E1 16363.634,E2 16363.634} C_VEL
LIN {X 0,Y 269.352,Z 580.66,A -85,B 0,C 180,E1 16371.861,E2 16371.861} C_VEL
LIN {X 0,Y 270.289,Z 580.66,A -85,B 0,C 180,E1 16379.991,E2 16379.991} C_VEL
LIN {X 0,Y 269.636,Z 580.66,A -85,B 0,C 180,E1 16386.439,E2 16386.439} C_VEL
LIN {X 0,Y 269.105,Z 580.66,A -85,B 0,C 180,E1 16392.996,E2 16392.996} C_VEL
LIN {X 0,Y 268.642,Z 580.66,A -85,B 0,C 180,E1 16399.755,E2 16399.755} C_VEL
LIN {X 0,Y 268.278,Z 581.235,A -85,B 0,C 180,E1 16405.396,E2 16405.396} C_VEL
LIN {X 0,Y 270.776,Z 586.44,A -85,B 0,C 180,E1 16406.642,E2 16406.642} C_VEL
LIN {X 0,Y 273.356,Z 589.519,A -85,B 0,C 180,E1 16407.734,E2 16407.734} C_VEL
LIN {X 0,Y 287.45,Z 610.807,A -85,B 0,C 180,E1 16413.115,E2 16413.115} C_VEL
LIN {X 0,Y 301.007,Z 635.33,A -85,B 0,C 180,E1 16417.798,E2 16417.798} C_VEL
LIN {X 0,Y 312.334,Z 664.82,A -85,B 0,C 180,E1 16422.277,E2 16422.277} C_VEL
LIN {X 0,Y 315.115,Z 675.766,A -85,B 0,C 180,E1 16423.754,E2 16423.754} C_VEL
LIN {X 0,Y 306.536,Z 710.544,A -85,B 0,C 180,E1 16426.494,E2 16426.494} C_VEL
LIN {X 0,Y 297.018,Z 742.302,A -85,B 0,C 180,E1 16430.296,E2 16430.296} C_VEL
LIN {X 0,Y 287.807,Z 770.303,A -85,B 0,C 180,E1 16435.101,E2 16435.101} C_VEL
LIN {X 0,Y 279.653,Z 795.606,A -85,B 0,C 180,E1 16441.28,E2 16441.28} C_VEL
LIN {X 0,Y 274.416,Z 815.15,A -85,B 0,C 180,E1 16448.108,E2 16448.108} C_VEL
LIN {X 0,Y 272.14,Z 829.566,A -85,B 0,C 180,E1 16455.499,E2 16455.499} C_VEL
LIN {X 0,Y 272.053,Z 837.373,A -85,B 0,C 180,E1 16462,E2 16462} C_VEL
LIN {X 0,Y 272.318,Z 840.316,A -85,B 0,C 180,E1 16466.81,E2 16466.81} C_VEL
LIN {X 0,Y 272.495,Z 840.895,A -85,B 0,C 180,E1 16470.551,E2 16470.551} C_VEL
LIN {X 0,Y 272.172,Z 838.663,A -85,B 0,C 180,E1 16476.385,E2 16476.385} C_VEL
LIN {X 0,Y 272.046,Z 831.959,A -85,B 0,C 180,E1 16482.859,E2 16482.859} C_VEL
LIN {X 0,Y 273.627,Z 818.943,A -85,B 0,C 180,E1 16490.251,E2 16490.251} C_VEL
LIN {X 0,Y 278.447,Z 799.628,A -85,B 0,C 180,E1 16497.524,E2 16497.524} C_VEL
LIN {X 0,Y 286.02,Z 775.756,A -85,B 0,C 180,E1 16503.763,E2 16503.763} C_VEL
LIN {X 0,Y 295.644,Z 746.675,A -85,B 0,C 180,E1 16509.093,E2 16509.093} C_VEL
LIN {X 0,Y 305.179,Z 715.565,A -85,B 0,C 180,E1 16513.008,E2 16513.008} C_VEL
LIN {X 0,Y 313.976,Z 681.086,A -85,B 0,C 180,E1 16515.935,E2 16515.935} C_VEL
LIN {X 0,Y 315.061,Z 674.46,A -85,B 0,C 180,E1 16516.41,E2 16516.41} C_VEL
LIN {X 0,Y 305.334,Z 644.969,A -85,B 0,C 180,E1 16520.681,E2 16520.681} C_VEL
LIN {X 0,Y 291.525,Z 617.129,A -85,B 0,C 180,E1 16525.556,E2 16525.556} C_VEL
LIN {X 0,Y 283.106,Z 604.082,A -85,B 0,C 180,E1 16528.496,E2 16528.496} C_VEL
LIN {X 0,Y 277.175,Z 598.59,A -85,B 0,C 180,E1 16530.59,E2 16530.59} C_VEL
LIN {X 0,Y 267.141,Z 592.113,A -85,B 0,C 180,E1 16534.518,E2 16534.518} C_VEL
LIN {X 0,Y 264.248,Z 587.426,A -85,B 0,C 180,E1 16535.979,E2 16535.979} C_VEL
LIN {X 0,Y 260.659,Z 582.497,A -85,B 0,C 180,E1 16537.89,E2 16537.89} C_VEL
LIN {X 0,Y 260.45,Z 580.66,A -85,B 0,C 180,E1 16538.275,E2 16538.275} C_VEL
LIN {X 0,Y 261.074,Z 580.66,A -85,B 0,C 180,E1 16546.596,E2 16546.596} C_VEL
LIN {X 0,Y 261.651,Z 580.66,A -85,B 0,C 180,E1 16553.364,E2 16553.364} C_VEL
LIN {X 0,Y 262.388,Z 580.66,A -85,B 0,C 180,E1 16560.009,E2 16560.009} C_VEL
LIN {X 0,Y 261.679,Z 580.66,A -85,B 0,C 180,E1 16566.654,E2 16566.654} C_VEL
LIN {X 0,Y 261.124,Z 580.66,A -85,B 0,C 180,E1 16573.42,E2 16573.42} C_VEL
LIN {X 0,Y 260.478,Z 580.66,A -85,B 0,C 180,E1 16581.575,E2 16581.575} C_VEL
LIN {X 0,Y 260.206,Z 581.216,A -85,B 0,C 180,E1 16587.831,E2 16587.831} C_VEL
LIN {X 0,Y 262.425,Z 586.279,A -85,B 0,C 180,E1 16589.221,E2 16589.221} C_VEL
LIN {X 0,Y 265.109,Z 589.199,A -85,B 0,C 180,E1 16590.623,E2 16590.623} C_VEL
LIN {X 0,Y 276.841,Z 608.341,A -85,B 0,C 180,E1 16596.75,E2 16596.75} C_VEL
LIN {X 0,Y 287.446,Z 630.598,A -85,B 0,C 180,E1 16602.494,E2 16602.494} C_VEL
LIN {X 0,Y 294.588,Z 653.289,A -85,B 0,C 180,E1 16607.633,E2 16607.633} C_VEL
LIN {X 0,Y 297.95,Z 675.287,A -85,B 0,C 180,E1 16612.43,E2 16612.43} C_VEL
LIN {X 0,Y 298.004,Z 684.349,A -85,B 0,C 180,E1 16614.393,E2 16614.393} C_VEL
LIN {X 0,Y 288.441,Z 708.901,A -85,B 0,C 180,E1 16619.221,E2 16619.221} C_VEL
LIN {X 0,Y 279.395,Z 729.399,A -85,B 0,C 180,E1 16625.171,E2 16625.171} C_VEL
LIN {X 0,Y 272.076,Z 744.917,A -85,B 0,C 180,E1 16632.181,E2 16632.181} C_VEL
LIN {X 0,Y 268.167,Z 753.591,A -85,B 0,C 180,E1 16638.606,E2 16638.606} C_VEL
LIN {X 0,Y 266.069,Z 758.684,A -85,B 0,C 180,E1 16646.741,E2 16646.741} C_VEL
LIN {X 0,Y 266.134,Z 758.637,A -85,B 0,C 180,E1 16653.264,E2 16653.264} C_VEL
LIN {X 0,Y 267.515,Z 754.965,A -85,B 0,C 180,E1 16659.778,E2 16659.778} C_VEL
LIN {X 0,Y 271.547,Z 746.065,A -85,B 0,C 180,E1 16667.024,E2 16667.024} C_VEL
LIN {X 0,Y 278.528,Z 731.114,A -85,B 0,C 180,E1 16674.063,E2 16674.063} C_VEL
LIN {X 0,Y 287.303,Z 711.475,A -85,B 0,C 180,E1 16680.045,E2 16680.045} C_VEL
LIN {X 0,Y 296.819,Z 687.261,A -85,B 0,C 180,E1 16685.006,E2 16685.006} C_VEL
LIN {X 0,Y 298.232,Z 680.697,A -85,B 0,C 180,E1 16686.231,E2 16686.231} C_VEL
LIN {X 0,Y 295.412,Z 657.659,A -85,B 0,C 180,E1 16691.296,E2 16691.296} C_VEL
LIN {X 0,Y 289.114,Z 635.265,A -85,B 0,C 180,E1 16696.273,E2 16696.273} C_VEL
LIN {X 0,Y 278.836,Z 611.805,A -85,B 0,C 180,E1 16702.092,E2 16702.092} C_VEL
LIN {X 0,Y 267.664,Z 593.541,A -85,B 0,C 180,E1 16707.779,E2 16707.779} C_VEL
LIN {X 0,Y 263.87,Z 587.438,A -85,B 0,C 180,E1 16709.864,E2 16709.864} C_VEL
LIN {X 0,Y 260.421,Z 582.861,A -85,B 0,C 180,E1 16711.735,E2 16711.735} C_VEL
LIN {X 0,Y 260.147,Z 580.66,A -85,B 0,C 180,E1 16712.241,E2 16712.241} C_VEL
LIN {X 0,Y 260.594,Z 580.66,A -85,B 0,C 180,E1 16719.589,E2 16719.589} C_VEL
LIN {X 0,Y 261.038,Z 580.66,A -85,B 0,C 180,E1 16726.576,E2 16726.576} C_VEL
LIN {X 0,Y 261.671,Z 580.66,A -85,B 0,C 180,E1 16733.346,E2 16733.346} C_VEL
LIN {X 0,Y 262.381,Z 580.66,A -85,B 0,C 180,E1 16739.991,E2 16739.991} C_VEL
LIN {X 0,Y 261.688,Z 580.66,A -85,B 0,C 180,E1 16746.635,E2 16746.635} C_VEL
LIN {X 0,Y 261.135,Z 580.66,A -85,B 0,C 180,E1 16753.4,E2 16753.4} C_VEL
LIN {X 0,Y 260.474,Z 581.07,A -85,B 0,C 180,E1 16762.045,E2 16762.045} C_VEL
LIN {X 0,Y 262.703,Z 586.185,A -85,B 0,C 180,E1 16763.377,E2 16763.377} C_VEL
LIN {X 0,Y 265.595,Z 589.193,A -85,B 0,C 180,E1 16764.784,E2 16764.784} C_VEL
LIN {X 0,Y 278.957,Z 609.083,A -85,B 0,C 180,E1 16770.575,E2 16770.575} C_VEL
LIN {X 0,Y 292.578,Z 632.714,A -85,B 0,C 180,E1 16775.707,E2 16775.707} C_VEL
LIN {X 0,Y 303.912,Z 660.312,A -85,B 0,C 180,E1 16780.353,E2 16780.353} C_VEL
LIN {X 0,Y 308.675,Z 678.204,A -85,B 0,C 180,E1 16782.929,E2 16782.929} C_VEL
LIN {X 0,Y 299.75,Z 712.254,A -85,B 0,C 180,E1 16785.757,E2 16785.757} C_VEL
LIN {X 0,Y 289.834,Z 743.688,A -85,B 0,C 180,E1 16789.671,E2 16789.671} C_VEL
LIN {X 0,Y 279.838,Z 772.607,A -85,B 0,C 180,E1 16794.908,E2 16794.908} C_VEL
LIN {X 0,Y 271.65,Z 796.953,A -85,B 0,C 180,E1 16801.265,E2 16801.265} C_VEL
LIN {X 0,Y 266.346,Z 815.875,A -85,B 0,C 180,E1 16808.313,E2 16808.313} C_VEL
LIN {X 0,Y 264.223,Z 829.574,A -85,B 0,C 180,E1 16815.902,E2 16815.902} C_VEL
LIN {X 0,Y 264.323,Z 837.448,A -85,B 0,C 180,E1 16823.419,E2 16823.419} C_VEL
LIN {X 0,Y 264.764,Z 839.775,A -85,B 0,C 180,E1 16829.997,E2 16829.997} C_VEL
LIN {X 0,Y 264.326,Z 837.464,A -85,B 0,C 180,E1 16836.575,E2 16836.575} C_VEL
LIN {X 0,Y 264.198,Z 830.731,A -85,B 0,C 180,E1 16843.248,E2 16843.248} C_VEL
LIN {X 0,Y 265.966,Z 817.735,A -85,B 0,C 180,E1 16850.838,E2 16850.838} C_VEL
LIN {X 0,Y 271.222,Z 798.351,A -85,B 0,C 180,E1 16858.323,E2 16858.323} C_VEL
LIN {X 0,Y 279.216,Z 774.444,A -85,B 0,C 180,E1 16864.702,E2 16864.702} C_VEL
LIN {X 0,Y 289.129,Z 745.861,A -85,B 0,C 180,E1 16870.034,E2 16870.034} C_VEL
LIN {X 0,Y 299.297,Z 714.108,A -85,B 0,C 180,E1 16874.068,E2 16874.068} C_VEL
LIN {X 0,Y 308.441,Z 679.621,A -85,B 0,C 180,E1 16876.992,E2 16876.992} C_VEL
LIN {X 0,Y 307.594,Z 672.681,A -85,B 0,C 180,E1 16877.838,E2 16877.838} C_VEL
LIN {X 0,Y 297.83,Z 644.119,A -85,B 0,C 180,E1 16882.304,E2 16882.304} C_VEL
LIN {X 0,Y 284.948,Z 618.431,A -85,B 0,C 180,E1 16887.238,E2 16887.238} C_VEL
LIN {X 0,Y 269.336,Z 594.415,A -85,B 0,C 180,E1 16893.543,E2 16893.543} C_VEL
LIN {X 0,Y 267.141,Z 592.113,A -85,B 0,C 180,E1 16894.518,E2 16894.518} C_VEL
LIN {X 0,Y 262.3,Z 588.939,A -85,B 0,C 180,E1 16896.73,E2 16896.73} C_VEL
LIN {X 0,Y 257.32,Z 587.873,A -85,B 0,C 180,E1 16899.141,E2 16899.141} C_VEL
LIN {X 0,Y 253.178,Z 583.329,A -85,B 0,C 180,E1 16901.712,E2 16901.712} C_VEL
LIN {X 0,Y 252.821,Z 580.66,A -85,B 0,C 180,E1 16902.362,E2 16902.362} C_VEL
LIN {X 0,Y 253.432,Z 580.66,A -85,B 0,C 180,E1 16909.685,E2 16909.685} C_VEL
LIN {X 0,Y 254.111,Z 580.66,A -85,B 0,C 180,E1 16916.594,E2 16916.594} C_VEL
LIN {X 0,Y 254.482,Z 580.66,A -85,B 0,C 180,E1 16920.01,E2 16920.01} C_VEL
LIN {X 0,Y 253.759,Z 580.66,A -85,B 0,C 180,E1 16926.863,E2 16926.863} C_VEL
LIN {X 0,Y 253.138,Z 580.66,A -85,B 0,C 180,E1 16933.852,E2 16933.852} C_VEL
LIN {X 0,Y 252.504,Z 580.66,A -85,B 0,C 180,E1 16942.292,E2 16942.292} C_VEL
LIN {X 0,Y 252.509,Z 581.171,A -85,B 0,C 180,E1 16943.712,E2 16943.712} C_VEL
LIN {X 0,Y 254.683,Z 586.29,A -85,B 0,C 180,E1 16945.412,E2 16945.412} C_VEL
LIN {X 0,Y 257.661,Z 589.224,A -85,B 0,C 180,E1 16947.212,E2 16947.212} C_VEL
LIN {X 0,Y 266.617,Z 603.64,A -85,B 0,C 180,E1 16952.628,E2 16952.628} C_VEL
LIN {X 0,Y 276.378,Z 621.615,A -85,B 0,C 180,E1 16958.176,E2 16958.176} C_VEL
LIN {X 0,Y 285.15,Z 644.362,A -85,B 0,C 180,E1 16963.962,E2 16963.962} C_VEL
LIN {X 0,Y 290.14,Z 666.106,A -85,B 0,C 180,E1 16968.994,E2 16968.994} C_VEL
LIN {X 0,Y 291.654,Z 685.652,A -85,B 0,C 180,E1 16973.495,E2 16973.495} C_VEL
LIN {X 0,Y 281.776,Z 710.131,A -85,B 0,C 180,E1 16978.41,E2 16978.41} C_VEL
LIN {X 0,Y 272.326,Z 730.6,A -85,B 0,C 180,E1 16984.481,E2 16984.481} C_VEL
LIN {X 0,Y 264.633,Z 746.112,A -85,B 0,C 180,E1 16991.663,E2 16991.663} C_VEL
LIN {X 0,Y 260.506,Z 754.78,A -85,B 0,C 180,E1 16998.266,E2 16998.266} C_VEL
LIN {X 0,Y 258.289,Z 759.867,A -85,B 0,C 180,E1 17006.643,E2 17006.643} C_VEL
LIN {X 0,Y 258.353,Z 759.822,A -85,B 0,C 180,E1 17013.363,E2 17013.363} C_VEL
LIN {X 0,Y 259.807,Z 756.157,A -85,B 0,C 180,E1 17020.072,E2 17020.072} C_VEL
LIN {X 0,Y 264.08,Z 747.258,A -85,B 0,C 180,E1 17027.52,E2 17027.52} C_VEL
LIN {X 0,Y 271.422,Z 732.318,A -85,B 0,C 180,E1 17034.734,E2 17034.734} C_VEL
LIN {X 0,Y 280.574,Z 712.721,A -85,B 0,C 180,E1 17040.841,E2 17040.841} C_VEL
LIN {X 0,Y 290.476,Z 688.541,A -85,B 0,C 180,E1 17045.887,E2 17045.887} C_VEL
